(* IEC 61131-3 sources: elnaProjects/ElpcLogic/PomarKc7Changed/build_USO_ecl (part 3) *)

  IM_SingleSignals_dP_maslo_gaz_Less100_status := DWORD_TO_UDINT(Im.SingleSignals.dP_maslo_gaz_Less100.status);

  IM_SingleSignals_dp_kran1_Less100_status := DWORD_TO_UDINT(Im.SingleSignals.dp_kran1_Less100.status);

  IM_SingleSignals_Razreshenie_zagruzki_dvig_status := DWORD_TO_UDINT(Im.SingleSignals.Razreshenie_zagruzki_dvig.status);

  IM_SingleSignals_Vozbud_gotovnost_status := DWORD_TO_UDINT(Im.SingleSignals.Vozbud_gotovnost.status);

  IM_SingleSignals_Vozbud_neispr_tsepey_upr_AVR_pit_status := DWORD_TO_UDINT(Im.SingleSignals.Vozbud_neispr_tsepey_upr_AVR_pit.status);

  IM_SingleSignals_Vozbud_neispravnost_status := DWORD_TO_UDINT(Im.SingleSignals.Vozbud_neispravnost.status);

  IM_SingleSignals_SHAVR1_v_rabote_status := DWORD_TO_UDINT(Im.SingleSignals.SHAVR1_v_rabote.status);

  IM_SingleSignals_SHAVR2_v_rabote_status := DWORD_TO_UDINT(Im.SingleSignals.SHAVR2_v_rabote.status);

  IM_SingleSignals_Avariinoe_otkluch_vikluchatelya_status := DWORD_TO_UDINT(Im.SingleSignals.Avariinoe_otkluch_vikluchatelya.status);

  IM_SingleSignals_Assinhronnii_hod_peregruzka_status := DWORD_TO_UDINT(Im.SingleSignals.Assinhronnii_hod_peregruzka.status);

  IM_SingleSignals_SHU_v_GPA_vkluch_status := DWORD_TO_UDINT(Im.SingleSignals.SHU_v_GPA_vkluch.status);

  IM_SingleSignals_SHP_v_GPA_vkluch_status := DWORD_TO_UDINT(Im.SingleSignals.SHP_v_GPA_vkluch.status);

  IM_SingleSignals_QF1_on_status := DWORD_TO_UDINT(Im.SingleSignals.QF1_on.status);

  IM_SingleSignals_QF2_on_status := DWORD_TO_UDINT(Im.SingleSignals.QF2_on.status);

  IM_SingleSignals_QF23_on_status := DWORD_TO_UDINT(Im.SingleSignals.QF23_on.status);

  IM_SingleSignals_QF4_QF5_on_status := DWORD_TO_UDINT(Im.SingleSignals.QF4_QF5_on.status);

  IM_SingleSignals_QF6_QF7_on_status := DWORD_TO_UDINT(Im.SingleSignals.QF6_QF7_on.status);

  IM_SingleSignals_QF8_QF9_on_status := DWORD_TO_UDINT(Im.SingleSignals.QF8_QF9_on.status);

  IM_SingleSignals_QF10_QF11_on_status := DWORD_TO_UDINT(Im.SingleSignals.QF10_QF11_on.status);

  IM_SingleSignals_QF12_QF13_on_status := DWORD_TO_UDINT(Im.SingleSignals.QF12_QF13_on.status);

  IM_SingleSignals_QF14_QF15_on_status := DWORD_TO_UDINT(Im.SingleSignals.QF14_QF15_on.status);

  IM_SingleSignals_QF22_on_status := DWORD_TO_UDINT(Im.SingleSignals.QF22_on.status);

  IM_SingleSignals_NS_G1_G2_status := DWORD_TO_UDINT(Im.SingleSignals.NS_G1_G2.status);

  IM_SingleSignals_NS_G3_G4_status := DWORD_TO_UDINT(Im.SingleSignals.NS_G3_G4.status);

  IM_SingleSignals_NS_G15_G16_status := DWORD_TO_UDINT(Im.SingleSignals.NS_G15_G16.status);

  IM_SingleSignals_NS_G17_status := DWORD_TO_UDINT(Im.SingleSignals.NS_G17.status);

  IM_SingleSignals_NS_G5_G6_status := DWORD_TO_UDINT(Im.SingleSignals.NS_G5_G6.status);

  IM_SingleSignals_NS_G7_G8_status := DWORD_TO_UDINT(Im.SingleSignals.NS_G7_G8.status);

  IM_SingleSignals_NS_G18_G19_status := DWORD_TO_UDINT(Im.SingleSignals.NS_G18_G19.status);

  IM_SingleSignals_NS_G10_G11_status := DWORD_TO_UDINT(Im.SingleSignals.NS_G10_G11.status);

  IM_SingleSignals_NS_G13_G14_status := DWORD_TO_UDINT(Im.SingleSignals.NS_G13_G14.status);

  IM_SingleSignals_Uroven_masla_akkum_status := DWORD_TO_UDINT(Im.SingleSignals.Uroven_masla_akkum.status);

  IM_SingleSignals_NKU1_GPA_on_status := DWORD_TO_UDINT(Im.SingleSignals.NKU1_GPA_on.status);

  IM_SingleSignals_NKU2_GPA_on_status := DWORD_TO_UDINT(Im.SingleSignals.NKU2_GPA_on.status);

  IM_SingleSignals_AO_KC_ot_SHKS_status := DWORD_TO_UDINT(Im.SingleSignals.AO_KC_ot_SHKS.status);

  IM_SingleSignals_AO_GPA_ot_SHU_status := DWORD_TO_UDINT(Im.SingleSignals.AO_GPA_ot_SHU.status);

  IM_SingleSignals_BEAO_srabotal_status := DWORD_TO_UDINT(Im.SingleSignals.BEAO_srabotal.status);

  IM_SingleSignals_Chastotny_pusk_status := DWORD_TO_UDINT(Im.SingleSignals.Chastotny_pusk.status);

  IM_SingleSignals_Neuspesh_chastotny_pusk_status := DWORD_TO_UDINT(Im.SingleSignals.Neuspesh_chastotny_pusk.status);

  IM_SingleSignals_Rezhim_ruchnogo_regulirovaniya_status := DWORD_TO_UDINT(Im.SingleSignals.Rezhim_ruchnogo_regulirovaniya.status);

  IM_SingleSignals_Osnovnoy_regul_off_status := DWORD_TO_UDINT(Im.SingleSignals.Osnovnoy_regul_off.status);

  IM_SingleSignals_Voltage_sekcii_norm_status := DWORD_TO_UDINT(Im.SingleSignals.Voltage_sekcii_norm.status);

  IM_SingleSignals_Reactorny_pusk_status := DWORD_TO_UDINT(Im.SingleSignals.Reactorny_pusk.status);

  IM_SingleSignals_NO_GPA_ot_SHU_status := DWORD_TO_UDINT(Im.SingleSignals.NO_GPA_ot_SHU.status);

  IM_SingleSignals_AO_GPA_ot_PRU_status := DWORD_TO_UDINT(Im.SingleSignals.AO_GPA_ot_PRU.status);

  IM_SingleSignals_Nalichie_BP1_status := DWORD_TO_UDINT(Im.SingleSignals.Nalichie_BP1.status);

  IM_SingleSignals_Nalichie_BP2_status := DWORD_TO_UDINT(Im.SingleSignals.Nalichie_BP2.status);

  IM_SingleSignals_Nalichie_BP3_status := DWORD_TO_UDINT(Im.SingleSignals.Nalichie_BP3.status);

  IM_SingleSignals_Nalichie_BP4_status := DWORD_TO_UDINT(Im.SingleSignals.Nalichie_BP4.status);

  IM_SingleSignals_Nalichie_BP5_status := DWORD_TO_UDINT(Im.SingleSignals.Nalichie_BP5.status);

  IM_SingleSignals_Nalichie_BP6_status := DWORD_TO_UDINT(Im.SingleSignals.Nalichie_BP6.status);

  IM_SingleSignals_Nalichie_BP7_BP8_status := DWORD_TO_UDINT(Im.SingleSignals.Nalichie_BP7_BP8.status);

  IM_SingleSignals_Nalichie_BP9_BP10_status := DWORD_TO_UDINT(Im.SingleSignals.Nalichie_BP9_BP10.status);

  IM_SingleSignals_Nalichie_cepei_upravlen_mv_status := DWORD_TO_UDINT(Im.SingleSignals.Nalichie_cepei_upravlen_mv.status);

  IM_SingleSignals_Nalichie_220BEAO_status := DWORD_TO_UDINT(Im.SingleSignals.Nalichie_220BEAO.status);

  IM_SingleSignals_Nalichie_per_220_na_vhode_status := DWORD_TO_UDINT(Im.SingleSignals.Nalichie_per_220_na_vhode.status);

  IM_SingleSignals_Nalichie_post_220_na_vhode_status := DWORD_TO_UDINT(Im.SingleSignals.Nalichie_post_220_na_vhode.status);

  IM_SingleSignals_Nalichie_BP11_status := DWORD_TO_UDINT(Im.SingleSignals.Nalichie_BP11.status);

  IM_SingleSignals_Nalichie_BP12_status := DWORD_TO_UDINT(Im.SingleSignals.Nalichie_BP12.status);

  IM_SingleSignals_Dver_SHU_pered_otkrita_status := DWORD_TO_UDINT(Im.SingleSignals.Dver_SHU_pered_otkrita.status);

  IM_SingleSignals_Dver_SHU_zad_otkrita_status := DWORD_TO_UDINT(Im.SingleSignals.Dver_SHU_zad_otkrita.status);

  IM_SingleSignals_EO_GPA_ot_knopki_SHU_status := DWORD_TO_UDINT(Im.SingleSignals.EO_GPA_ot_knopki_SHU.status);

  IM_SingleSignals_EO_EGPA_ot_PRY_status := DWORD_TO_UDINT(Im.SingleSignals.EO_EGPA_ot_PRY.status);

  IM_SingleSignals_Synchroniz_rezhima_K1_status := DWORD_TO_UDINT(Im.SingleSignals.Synchroniz_rezhima_K1.status);

  IM_SingleSignals_Potok_ms_posle_AVOM_status := DWORD_TO_UDINT(Im.SingleSignals.Potok_ms_posle_AVOM.status);

  IM_Kran1_status := DWORD_TO_UDINT(Im.Kran1.status);

  IM_Kran2_status := DWORD_TO_UDINT(Im.Kran2.status);

  IM_Kran3_status := DWORD_TO_UDINT(Im.Kran3.status);

  IM_Kran3b_status := DWORD_TO_UDINT(Im.Kran3b.status);

  IM_Kran4_status := DWORD_TO_UDINT(Im.Kran4.status);

  IM_Kran5_status := DWORD_TO_UDINT(Im.Kran5.status);

  IM_Kran6_status := DWORD_TO_UDINT(Im.Kran6.status);

  IM_nu1_status := DWORD_TO_UDINT(Im.nu1.status);

  IM_nu2_status := DWORD_TO_UDINT(Im.nu2.status);

  IM_pns_status := DWORD_TO_UDINT(Im.pns.status);

  IM_v1_Avom_status := DWORD_TO_UDINT(Im.v1_Avom.status);

  IM_v2_Avom_status := DWORD_TO_UDINT(Im.v2_Avom.status);

  IM_v3_Avom_status := DWORD_TO_UDINT(Im.v3_Avom.status);

  IM_v4_Avom_status := DWORD_TO_UDINT(Im.v4_Avom.status);

  IM_mv_status := DWORD_TO_UDINT(Im.mv.status);

  IM_KaloriferAVOM_status := DWORD_TO_UDINT(Im.KaloriferAVOM.status);

  IM_CMN_status := DWORD_TO_UDINT(Im.CMN.status);

  IM_TEN_kollectora_status := DWORD_TO_UDINT(Im.TEN_kollectora.status);

  IM_TEN_MB_status := DWORD_TO_UDINT(Im.TEN_MB.status);
END_FUNCTION_BLOCK

FUNCTION_BLOCK fb_RashodAlg
  VAR_INPUT
    P_gasIn : struct_AI;
  END_VAR
  VAR_IN_OUT
    StrAi : struct_AI;
  END_VAR
  VAR_INPUT
    T_gasIn : struct_AI;
    dP_konf : struct_AI;
    K : struct_AnalogParametr;
    A : struct_AnalogParametr;
    y0 : struct_AnalogParametr;
  END_VAR
  VAR
    num : LREAL;
    den : LREAL;
    _statusAi : TYPE_StatusAi;
  END_VAR
  VAR CONSTANT
    P0 : LREAL          := 0.1033;
    T0 : LREAL          := 293.0;
  END_VAR

  strAI.opcCommandsDisabled := strAI.inopcCommandsDisabled ;

  IF (P_gasIn.interval < _statusAi.normal) OR
     (T_gasIn.interval < _statusAi.normal) OR
     (dP_konf.interval < _statusAi.normal) THEN
  	StrAi.interval := _statusAi.NOTRELIABLE;
            strAI.status := 	SHL(BOOL_TO_DWORD(strAI.OpcCommandsDisabled ), 21)
  	OR BYTE_TO_DWORD(strAI.interval);
  	RETURN;
  END_IF;

  IF (P_gasIn.value <0.3) THEN
  	StrAi.interval := _statusAi.normal;
  	StrAi.value:= 0.0;
            strAI.status := 	SHL(BOOL_TO_DWORD(strAI.OpcCommandsDisabled ), 21)
  	OR BYTE_TO_DWORD(strAI.interval);
  	RETURN;
  END_IF;

  StrAi.interval:= _statusAi.normal;

  num:= (dP_konf.Value/1000.0)*(T_gasIn.value+273.0)*P0*735.56*K.Value;
  den:= y0.Value*P_gasIn.value*T0 ;

  StrAi.value:= A.Value*SQRT(num/den);

  strAI.status := 	SHL(BOOL_TO_DWORD(strAI.OpcCommandsDisabled ), 21) (* Управление в ВУ заблокировано *)
  		OR BYTE_TO_DWORD(strAI.interval);	              (* интервал *)
END_FUNCTION_BLOCK

FUNCTION_BLOCK fb_Question
  VAR_IN_OUT
    StrQ : struct_Question;
  END_VAR
  VAR
    Asked : UINT;
    _answers : TYPE_Answers;
    _sunpackerCommand : fb_sunpackerCommand;
    source : BYTE;
    parametr : BYTE;
    lastParametr : BYTE;
    cmd : BYTE;
    source_for_Status : BYTE;
    cmd_for_Status : BYTE;
    command_error_for_Status : BYTE;
    resetCmdTimer : TON;
    resetCmdTimerPriznak : BOOL;
    reset_Trig : R_TRIG;
  END_VAR
  VAR CONSTANT
    cmd_answer : UINT          := 1;
  END_VAR

  StrQ.OpcCommandsDisabled := StrQ.inopcCommandsDisabled;

  IF StrQ.ask THEN
  StrQ.inopcCommandsDisabled:=FALSE;
      IF Asked=0 THEN
  	Asked:=StrQ.AnswerVariants;
  	StrQ.answer:=_answers.ANS_NONE;
      END_IF;

      _sunpackerCommand(command := StrQ.inCommand);
  	source := _sunpackerCommand.source;
            parametr := _sunpackerCommand.parametr;
  	cmd := _sunpackerCommand.cmd;

      IF cmd <> 0 AND lastParametr <> parametr AND ((NOT StrQ.OpcCommandsDisabled) AND source > 0)  then
  	CASE BYTE_TO_INT(cmd) OF
  	                               1 :

  				IF Asked<>0 THEN
                                             (* CASE BYTE_TO_INT(parametr) OF
                                              1: answer:=_answers.ANS_YES;
                                              2: answer:=_answers.ANS_NO;
                                              4: answer:=_answers.ANS_CANCEL;
                                              8: answer:=_answers.ANS_RETRY;
  	                                  END_CASE;*)
                                          StrQ.answer:=BYTE_TO_UINT(parametr);
                                          command_error_for_Status := 0;
                                          ELSE
  	                              command_error_for_Status := cmd;
                                          END_IF;
  	END_CASE;
  	source_for_Status := source;
  	cmd_for_Status := cmd;
  	resetCmdTimer(IN := FALSE);
  	resetCmdTimerPriznak := TRUE;
      END_IF;

      lastParametr := parametr;

      resetCmdTimer(IN := resetCmdTimerPriznak, PT := T#5S);
      IF resetCmdTimer.Q THEN
  	resetCmdTimerPriznak := FALSE;
  	source_for_Status := 0;
  	cmd_for_Status := 0;
  	command_error_for_Status := 0;
      END_IF;
  END_IF;

  reset_Trig(CLK := StrQ.reset);
  IF reset_Trig.Q THEN
  	Asked:=0;
  	StrQ.answer:=0;
            StrQ.ask:=FALSE;
            StrQ.reset:=FALSE;
  	StrQ.inopcCommandsDisabled:=TRUE;
  END_IF;

  StrQ.status := SHL(BYTE_TO_DWORD(source_for_Status), 29)
  			OR SHL(BYTE_TO_DWORD(cmd_for_Status), 26)
  			OR SHL(BYTE_TO_DWORD(command_error_for_Status), 23)
  			OR SHL(BOOL_TO_DWORD(StrQ.OpcCommandsDisabled ), 21);
  IF StrQ.answer = 0 THEN
      StrQ.status := StrQ.status  OR SHL(UINT_TO_DWORD(asked), 6);
  ELSE
      StrQ.status := StrQ.status  OR SHL(UINT_TO_DWORD(StrQ.answer), 6);
  END_IF;
END_FUNCTION_BLOCK

FUNCTION_BLOCK fb_ph_AIprotection
  VAR_IN_OUT
    StrAiP : struct_AiProtection;
  END_VAR
  VAR_INPUT
    act : TYPE_PhaseAlgoritmAction;
    PhaseNumber : UINT;
  END_VAR
  VAR_IN_OUT
    StrPh : struct_PhaseAlgoritm;
  END_VAR
  VAR
    CommandFault_Trig : R_TRIG;
    reset_Trig : R_TRIG;
    _statusDualInput : TYPE_statusDualInput;
  END_VAR

  IF StrPh.run AND NOT StrPh.start THEN
  	StrPh.start := TRUE;
  	StrPh.top := FALSE;
  	StrPh.error := FALSE;
            StrPh.run:=FALSE;

  	CASE act OF
  		(*PhaseAlgoritmAction.run*)    _run : runAiProtection(StrAiP); (*cmd_run*)
  		(*PhaseAlgoritmAction.reset*)_reset : resetAiProtection(StrAiP); (*cmd_reset*)
  	END_CASE;
  END_IF;

  IF StrPh.start AND NOT StrPh.top THEN
                      CommandFault_Trig(CLK := StrAiP.hasError);
                      IF CommandFault_Trig.Q THEN
  	          StrPh.error := TRUE;
                      END_IF;

  		CASE act OF
  		(*PhaseAlgoritmAction.run*)    _run:    StrPh.top:=StrAiP.isRunning;

  		(*PhaseAlgoritmAction.reset*) _reset:   StrPh.top := NOT StrAiP.isRunning;
  		END_CASE;

  END_IF;

  IF StrPh.top THEN
  StrPh.error := FALSE;
  END_IF;

  reset_Trig(CLK := StrPh.reset);
  IF reset_Trig.Q THEN
            StrPh.start := FALSE;
  	StrPh.error := FALSE;
  	StrPh.top := FALSE;
            StrPh.run:=FALSE;
            StrPh.reset:=FALSE;
  END_IF;

  StrPh.startStatus := SHL(BOOL_TO_DWORD(StrPh.start), PhaseNumber);
  StrPh.errorStatus := SHL(BOOL_TO_DWORD(StrPh.error), PhaseNumber);
  StrPh.topStatus := SHL(BOOL_TO_DWORD(StrPh.top), PhaseNumber);
END_FUNCTION_BLOCK

FUNCTION_BLOCK fb_OilPump_Init
  VAR_INPUT
    data_Ini : BOOL;
    ISVALIDREF_statOn : BOOL;
    ISVALIDREF_statOff : BOOL;
    ISVALIDREF_cmdOn : BOOL;
    ISVALIDREF_cmdOff : BOOL;
    ISVALIDREF_inBreakCmdOn : BOOL;
    ISVALIDREF_inBreakCmdOff : BOOL;
  END_VAR
  VAR_IN_OUT
    str_Op : struct_OilPump;
  END_VAR
  VAR_OUTPUT
    Init : BOOL          := FALSE;
  END_VAR

  (*****            Функциональный блок переинициализации структуры  НУ          *****)

   Init := FALSE;

      IF data_Ini THEN                            (* Параметрам требуется переинициализация. *)
          str_Op.ISVALIDREF_statOn                := ISVALIDREF_statOn;
          str_Op.ISVALIDREF_statOff               := ISVALIDREF_statOff;
          str_Op.ISVALIDREF_cmdOn                 := ISVALIDREF_cmdOn;
          str_Op.ISVALIDREF_cmdOff                := ISVALIDREF_cmdOff;
          str_Op.ISVALIDREF_inBreakCmdOn          := ISVALIDREF_inBreakCmdOn;
          str_Op.ISVALIDREF_inBreakCmdOff         := ISVALIDREF_inBreakCmdOff;
          data_Ini:=FALSE;
          Init := TRUE;
      END_IF;

          ISVALIDREF_statOn:= FALSE;
          ISVALIDREF_statOff:= FALSE;
          ISVALIDREF_cmdOn:= FALSE;
          ISVALIDREF_cmdOff:= FALSE;
          ISVALIDREF_inBreakCmdOn:= FALSE;
          ISVALIDREF_inBreakCmdOff:= FALSE;
END_FUNCTION_BLOCK

FUNCTION_BLOCK fb_DO_Init
  VAR_INPUT
    data_Ini : BOOL;
    imit : BOOL          := FALSE;
  END_VAR
  VAR_IN_OUT
    strDO : struct_DO;
  END_VAR
  VAR_OUTPUT
    Init : BOOL          := FALSE;
  END_VAR

  (*****            Функциональный блок переинициализации структуры-дескриптора канала дискретного ввода.            *****)
   Init := FALSE;

      IF data_Ini THEN                            (* Параметрам требуется переинициализация. *)
          strDO.imit       := imit;
          data_Ini:=FALSE;
          Init := TRUE;
      END_IF;
    IF Init THEN
  imit:=FALSE;
     END_IF;
END_FUNCTION_BLOCK

FUNCTION_BLOCK fb_DOSourceMlp
  VAR_IN_OUT
    arDout : TWordData;
  END_VAR
  VAR_INPUT
    err_mod : TItemDIN;
  END_VAR
  VAR_IN_OUT
    strDO : struct_DO;
  END_VAR
  VAR
    bitNumber : INT;
  END_VAR

  strDO.blConnect := ((UINT_TO_WORD(err_mod.wValue) = 20) and (UINT_TO_WORD(err_mod.wFlags) = 192));

  strDO.value:=0;

  FOR bitNumber:=0 TO 15 BY 1 DO
  	strDO.value:=strDO.value OR (SHL(BOOL_TO_WORD(strDO.bits[bitNumber]),bitNumber));
  END_FOR;

  IF NOT strDO.imit THEN
  	 arDout.wValue:= WORD_TO_UINT(strDO.value);
  END_IF;
END_FUNCTION_BLOCK

FUNCTION_BLOCK fb_AnalogParametr
  VAR_IN_OUT
    StrAP : struct_AnalogParametr;
  END_VAR
  VAR
    _sunpackerCommand : fb_sunpackerCommand;
    source : BYTE;
    cmd : BYTE;
    source_for_Status : BYTE;
    cmd_for_Status : BYTE;
    command_error_for_Status : BYTE;
    resetCmdTimer : TON;
    resetCmdTimerPriznak : BOOL;
    secondTact : BOOL;
    inp : LREAL;
    rABS : LREAL;
  END_VAR

  IF NOT secondTact THEN
  	StrAP.Value := StrAP.currentValue;
  	secondTact := true;
  END_IF;

  StrAP.OpcCommandsDisabled := StrAP.inOpcCommandsDisabled;

   (* ---- Если управление с ВУ заблокировано, то передаем команду из алгоритма ---- *)
  IF StrAP.inOpcCommandsDisabled THEN
  	StrAP.inCommand := StrAP.inCommand_Alg;
  ELSE (* иначе передаем команду с АРМа*)
  	StrAP.inCommand := StrAP.inCommand_ARM;
  END_IF;

  _sunpackerCommand(command := StrAP.inCommand);
  	source := _sunpackerCommand.source;
  	cmd := _sunpackerCommand.cmd;

  IF cmd <> 0 AND StrAP.newValue <> StrAP.Value and (((NOT StrAP.opcCommandsDisabled) AND source > 0) OR source = 0) then
  	CASE BYTE_TO_INT(cmd) OF
  	(*cmd_ChangeValue*) 1 :
  				StrAP.isValidValue := TRUE;
  				IF StrAP.minVal_ISVALIDREF AND StrAP.isValidValue THEN
  					IF StrAP.newValue < StrAP.minVal THEN
  						StrAP.isValidValue := FALSE;
  					END_IF;
  				END_IF;
  				IF StrAP.maxVal_ISVALIDREF AND StrAP.isValidValue THEN
  					IF StrAP.newValue > StrAP.maxVal THEN
  						StrAP.isValidValue := FALSE;
  					END_IF;
  				END_IF;
  				IF StrAP.maxStep_ISVALIDREF AND StrAP.isValidValue  THEN
  					inp := StrAP.Value - StrAP.newValue;
  					IF inp < 0.0 THEN
  						rABS := -inp;
  					ELSE
  						rABS := inp;
  					END_IF;
  					IF rABS > StrAP.maxStep THEN
  						StrAP.isValidValue := FALSE;
  					END_IF;
  				END_IF;
  				IF StrAP.isValidValue THEN
  					StrAP.Value := StrAP.newValue;
  					command_error_for_Status := 0;
  				ELSE
  					command_error_for_Status := cmd;
  				END_IF;
  	END_CASE;
  	source_for_Status := source;
  	cmd_for_Status := cmd;
  	resetCmdTimer(IN := FALSE);
  	resetCmdTimerPriznak := TRUE;
  END_IF;

  resetCmdTimer(IN := resetCmdTimerPriznak, PT := T#5S);
  IF resetCmdTimer.Q THEN
  	resetCmdTimerPriznak := FALSE;
  	source_for_Status := 0;
  	cmd_for_Status := 0;
  	command_error_for_Status := 0;
  END_IF;

  StrAP.status := SHL(BYTE_TO_DWORD(source_for_Status), 29)
  			OR SHL(BYTE_TO_DWORD(cmd_for_Status), 26)
  			OR SHL(BYTE_TO_DWORD(command_error_for_Status), 23)
  			OR SHL(BOOL_TO_DWORD(StrAP.OpcCommandsDisabled ), 21);
END_FUNCTION_BLOCK

FUNCTION_BLOCK fb_AI_Init
  VAR_INPUT
    data_Ini : BOOL;
    dLL : LREAL;
    dHL : LREAL;
    dLA : LREAL;
    dHA : LREAL;
    dLW : LREAL;
    dHW : LREAL;
    ISVALIDREF_LA : BOOL          := False;
    ISVALIDREF_HA : BOOL          := False;
    ISVALIDREF_LW : BOOL          := False;
    ISVALIDREF_HW : BOOL          := False;
    delayLA : TIME          := T#0S;
    delayLW : TIME          := T#0S;
    delayHW : TIME          := T#0S;
    delayHA : TIME          := T#0S;
    inpLL : LREAL          := 4000.0;
    inpHL : LREAL          := 20000.0;
    CurrentShotCircuit : LREAL          := 21000.0;
    CurrentBreakCircuit : LREAL          := 3700.0;
    dMaxChangeSpeed : LREAL;
    dMaxChangeSpeedDown : LREAL;
    histeresis : LREAL;
    aperturFilter : LREAL;
    exponentialFilter : LREAL;
    rassoglasovanie : LREAL;
    inOpcCommandsDisabled : BOOL;
  END_VAR
  VAR_IN_OUT
    strAI : struct_AI;
  END_VAR
  VAR_OUTPUT
    Init : BOOL          := FALSE;
  END_VAR

  (*****            Функциональный блок переинициализации структуры-дескриптора канала аналогового ввода.            *****)
       Init := false;

      IF data_Ini THEN                            (* Параметрам требуется переинициализация. *)
          strAI.dLL                := dLL;
          strAI.dHL                := dHL;
          strAI.dLA                := dLA;
          strAI.dHA                := dHA;
          strAI.dLW                := dLW;
          strAI.dHW                := dHW;
          strAI.ISVALIDREF_LA      := ISVALIDREF_LA;
          strAI.ISVALIDREF_HA      := ISVALIDREF_HA;
          strAI.ISVALIDREF_LW      := ISVALIDREF_LW;
          strAI.ISVALIDREF_HW      := ISVALIDREF_HW;
          strAI.delayLA            := delayLA;
          strAI.delayLW            := delayLW;
          strAI.delayHW            := delayHW;
          strAI.delayHA            := delayHA;
          strAI.inpLL              := inpLL;
          strAI.inpHL              := inpHL;
          strAI.CurrentShotCircuit := CurrentShotCircuit;
          strAI.CurrentBreakCircuit:= CurrentBreakCircuit;
          strAI.dMaxChangeSpeed     := dMaxChangeSpeed;
          strAI.dMaxChangeSpeedDown := dMaxChangeSpeedDown;
          strAI.histeresis         := histeresis;
          strAI.aperturFilter      := aperturFilter;
          strAI.exponentialFilter  := exponentialFilter;
          strAI.rassoglasovanie    := rassoglasovanie;
          strAI.rassoglasovanie    := rassoglasovanie;

          data_Ini:=false;
          Init := TRUE;
       END_IF;
    IF Init THEN
          dLL:= 0.0;
          dHL:= 0.0;
          dLA:= 0.0;
          dHA:= 0.0;
          dLW:= 0.0;
          dHW:= 0.0;
          inpLL:= 4000.0;
          inpHL:= 20000.0;
          CurrentShotCircuit:= 21000.0;
          CurrentBreakCircuit:= 3700.0;
          ISVALIDREF_LA:= false;
          ISVALIDREF_HA:= false;
          ISVALIDREF_LW:= false;
          ISVALIDREF_HW:= false;
          delayLA:= T#0S;
          delayLW:= T#0S;
          delayHW:= T#0S;
          delayHA:= T#0S;
          dMaxChangeSpeed:= 0.0;
          dMaxChangeSpeedDown:= 0.0;
          histeresis:= 0.0;
          aperturFilter:= 0.0;
          exponentialFilter:= 0.0;
          rassoglasovanie:= 0.0;
        END_IF;
END_FUNCTION_BLOCK

FUNCTION_BLOCK fb_AiSourceMlp_timer
  VAR_INPUT
    arAIN : TItemAIN;
    err_mod : TItemDIN;
  END_VAR
  VAR_IN_OUT
    strAI : struct_AI;
  END_VAR
  VAR
    _statusAi : TYPE_StatusAi;
    _commandAnalog : TYPE_CommandAnalog;
    _sunpackerCommand : fb_sunpackerCommand;
    _AnalogLimitFlags : TYPE_AnalogLimitFlags;
    notReliable : BOOL;
    _lastValue : LREAL;
    resetCmdTimer : TON;
    _LastValueTimer : TON;
    resetCmdTimerPriznak : BOOL;
    k : LREAL;
    b : LREAL;
    ap : LREAL;
    raznitsa : LREAL;
    rABS : LREAL;
    h : LREAL;
    mismatch : LREAL;
    parametr : BYTE;
    source : BYTE;
    cmd : BYTE;
    lastCmd : BYTE;
    source_for_Status : BYTE;
    cmd_for_Status : BYTE;
    command_error_for_Status : BYTE;
    secondTakt : BOOL;
    off_trig : R_TRIG;
    on_trig : R_TRIG;
    remont_trig : R_TRIG;
    LL_trig : R_TRIG;
    HL_trig : R_TRIG;
    Normal_trig : R_TRIG;
    Nedostover_trig : R_TRIG;
    timerLA : TON;
    timerHA : TON;
    timerLW : TON;
    timerHW : TON;
  END_VAR
  VAR RETAIN
    retainLL : LREAL;
    retainHL : LREAL;
    retainLA : LREAL;
    retainHA : LREAL;
    retainLW : LREAL;
    retainHW : LREAL;
  END_VAR

  strAI.opcCommandsDisabled := strAI.inopcCommandsDisabled ;

  (* ---- При первом пуске принимаем значение уставок ---- *)
  IF NOT secondTakt THEN
            IF (strAI.dLL <> retainLL) AND (retainLL <> 0.0) THEN  strAI.LL := retainLL;
            ELSE strAI.LL := strAI.dLL; END_IF;
  	IF (strAI.dHL <> retainHL) AND (retainHL <> 0.0) THEN  strAI.HL := retainHL;
            ELSE strAI.HL := strAI.dHL; END_IF;

            IF strAI.ISVALIDREF_HA AND (strAI.dHA <> retainHA) AND (retainHA <> 0.0) THEN  strAI.HA := retainHA;
            ELSE strAI.HA := strAI.dHA; END_IF;

            IF strAI.ISVALIDREF_LA AND (strAI.dLA <> retainLA) AND (retainLA <> 0.0) THEN  strAI.LA := retainLA;
            ELSE strAI.LA := strAI.dLA; END_IF;

            IF strAI.ISVALIDREF_HW AND (strAI.dHW <> retainHW) AND (retainHW <> 0.0) THEN  strAI.HW := retainHW;
            ELSE strAI.HW := strAI.dHW; END_IF;

            IF strAI.ISVALIDREF_LW AND (strAI.dLW <> retainLW) AND (retainLW <> 0.0) THEN  strAI.LW := retainLW;
            ELSE strAI.LW := strAI.dLW; END_IF;

  	secondTakt  := TRUE;
  END_IF;

  (* ---- пересчет тока в физ величину ---- *)
  k := (strAI.HL - strAI.LL)/(strAI.inpHl - strAI.inpLL);
  b := strAI.LL - k * strAI.inpLL;
  strAI.value := k * arAIN.dblValue + b;

  (* ---- определение обрыва и кз ----- *)

  strAI.blConnect := true;(*(UINT_TO_WORD(arAIN.wFlags) = 1472) and (UINT_TO_WORD(err_mod.wValue) = 20) and (UINT_TO_WORD(err_mod.wFlags) = 192); *)
  IF NOT strAI.blConnect THEN
      strAI.interval := _statusAi.NOTDEFINED;
  ELSIF ((arAIN.dblValue < strAI.currentBreakCircuit) AND (strAI.currentBreakCircuit > 0.0)) OR ((strAI.interval = _statusAi.LL) AND (arAIN.dblValue < (strAI.currentBreakCircuit + 100.0))) THEN
      strAI.interval := _statusAi.LL;
  ELSIF ((arAIN.dblValue > strAI.currentShotCircuit) AND (strAI.currentShotCircuit > 0.0)) OR ((strAI.interval = _statusAi.HL) AND (arAIN.dblValue > (strAI.currentShotCircuit - 100.0))) THEN
      strAI.interval := _statusAi.HL;
  ELSE
      strAI.interval := _statusAi.normal;
  END_IF;

  IF NOT strAI.imit THEN
  	(* Расчет апертурного фильтра*)
  	ap := strAI.aperturFilter * 0.01 * (strAI.HL - strAI.LL);
  	IF strAI.aperturFilter <> 0.0 THEN raznitsa := strAI.value- _lastValue;
  		IF 	raznitsa < 0.0 	THEN 	rABS := -raznitsa; 		ELSE 	rABS := raznitsa; 		END_IF;
  		IF 	rABS > ap 	THEN 	strAI.value := strAI.value;	ELSE 	strAI.value := _lastValue; 	END_IF;
  	END_IF;

  	(* Расчет экпоненциального фильтра*)
  	IF strAI.exponentialFilter <> 0.0 THEN strAI.value := (strAI.exponentialFilter * strAI.value) + ((1.0 - strAI.exponentialFilter) * _lastValue); END_IF;
  ELSE
  	strAI.interval := _statusAi.normal;
  END_IF;

  IF notReliable THEN strAI.interval := _statusAi.NOTRELIABLE; END_IF;

  IF NOT notReliable THEN
  	IF strAI.interval >= _statusAi.normal THEN
  		strAI.interval := _statusAi.NOTDEFINED;
  		h := strAI.histeresis* 0.01 * (strAI.HL-strAI.LL);
  		(*определение выхода за аппаратные границы вынесено в GetData.здесь только для нужд имитации*)
  		IF strAI.imit THEN
  			mismatch := strAI.rassoglasovanie * 0.01 * (strAI.HL - strAI.LL);
  			IF ( strAI.value < strAI.LL - mismatch)   THEN strAI.interval := _statusAi.LL;
  			ELSIF  (strAI.value > strAI.Hl + mismatch) THEN strAI.interval := _statusAi.HL; END_IF;
  		ELSE
  			strAI.interval := _statusAi.normal;
  			IF strAI.ISVALIDREF_LA AND NOT strAI.Disabled_LA AND (strAI.interval = _statusAi.normal) THEN
                                timerLA(IN:=(strAI.value  < strAI.LA) OR ((strAI.interval = _statusAi.LA)  AND ((strAI.value - h) < strAI.LA)), PT:=strAI.delayLA);
  				IF timerLA.Q  THEN
  					strAI.interval := _statusAi.LA;
  				END_IF;
  			END_IF;
  			IF strAI.ISVALIDREF_HA  AND NOT strAI.Disabled_HA AND (strAI.interval = _statusAi.normal)  THEN
                                timerHA(IN:=(strAI.value > strAI.HA) OR ((strAI.interval = _statusAi.HA)  AND ((strAI.value + h) > strAI.HA)), PT:=strAI.delayHA);
  				IF timerHA.Q  THEN
  					strAI.interval := _statusAi.HA;
  				END_IF;
  			END_IF;
  			IF strAI.ISVALIDREF_LW AND NOT strAI.Disabled_LW AND (strAI.interval = _statusAi.normal)  THEN
                                timerLW(IN:=(strAI.value < strAI.LW) OR ((strAI.interval = _statusAi.LW)  AND ((strAI.value - h) < strAI.LW)), PT:=strAI.delayLW);
  				IF timerLW.Q THEN
  					strAI.interval := _statusAi.LW;
  				END_IF;
  			END_IF;
  			IF strAI.ISVALIDREF_HW AND NOT strAI.Disabled_HW  AND (strAI.interval = _statusAi.normal) THEN
                                timerHW(IN:=(strAI.value > strAI.HW)  OR ((strAI.interval = _statusAi.HW)  AND ((strAI.value + h) > strAI.HW)), PT:=strAI.delayHW);
  				IF  timerHW.Q  THEN
  					strAI.interval := _statusAi.HW;
  				END_IF;
  			END_IF;
  		END_IF;
  	END_IF;
  ELSE
  	strAI.interval := _statusAi.NOTRELIABLE;
  END_IF;

  IF strAI.remont THEN strAI.interval := _statusAi.NOTDEFINED; END_IF;

  _sunpackerCommand(command := strAI.inCommand);
  	source := _sunpackerCommand.source;
  	parametr := _sunpackerCommand.parametr;
  	cmd := _sunpackerCommand.cmd;

  IF cmd <> 0 AND lastCmd <> cmd and (((NOT strAI.opcCommandsDisabled) AND source > 0) OR source = 0) then
  	CASE BYTE_TO_INT(cmd) OF
  	(*cmd_SetUstavki*) 1 :
  				IF ((parametr AND _AnalogLimitFlags.LL) <> 0)		             	THEN 	strAI.LL := strAI.dLL; retainLL:= strAI.LL; END_IF;
  				IF ((parametr AND _AnalogLimitFlags.HL) <> 0)		 	          THEN	strAI.HL := strAI.dHL; retainHL:= strAI.HL; END_IF;
  				IF ((parametr AND _AnalogLimitFlags.LA) <> 0) AND strAI.ISVALIDREF_LA 	THEN	strAI.LA := strAI.dLA; retainLA:= strAI.LA; END_IF;
  				IF ((parametr AND _AnalogLimitFlags.HA) <> 0) AND strAI.ISVALIDREF_HA 	THEN	strAI.HA := strAI.dHA; retainHA:= strAI.HA; END_IF;
  				IF ((parametr AND _AnalogLimitFlags.LW) <> 0) AND strAI.ISVALIDREF_LW 	THEN	strAI.LW := strAI.dLW; retainLW:= strAI.LW; END_IF;
  				IF ((parametr AND _AnalogLimitFlags.HW) <> 0) AND strAI.ISVALIDREF_HW 	THEN	strAI.HW := strAI.dHW; retainHW:= strAI.HW; END_IF;
  	(*cmd_SetRemont*) 2 :
  				strAI.remont := TRUE;
  	(*cmd_ResetRemont*) 3 :
  				strAI.remont := FALSE;
  	(*cmd_kvitNotReliable*) 4 :
  				notReliable := FALSE;
  	END_CASE;
  	source_for_Status := source;
  	cmd_for_Status := cmd;
  	command_error_for_Status := 0;
  	resetCmdTimer(IN := FALSE);
  	resetCmdTimerPriznak := TRUE;
  END_IF;
  lastCmd := cmd;

  resetCmdTimer(IN := resetCmdTimerPriznak, PT := T#5S);
  IF resetCmdTimer.Q THEN
  	resetCmdTimerPriznak := FALSE;
  	source_for_Status := 0;
  	cmd_for_Status := 0;
  	command_error_for_Status := 0;
  END_IF;

  strAI.NS_Min := (strAI.value < strAI.minValue) AND strAI.minValue_ISVALIDREF;
  strAI.NS_Max := (strAI.value > strAI.maxValue) AND strAI.maxValue_ISVALIDREF;

  strAI.NS := (strAI.interval <= _statusAi.normal) AND NOT strAI.remont;

  Normal_trig(CLK := strAI.interval >= _statusAi.normal);

  IF NOT Normal_trig.Q THEN
  	_LastValueTimer(PT := T#1S);
  	IF (strAI.value<>_lastValue) OR _LastValueTimer.Q THEN
  		IF (_LastValueTimer.ET>T#0MS) THEN
  			strAI.ChangeSpeed:=(strAI.value-_lastValue)/(TIME_TO_LREAL(_LastValueTimer.ET)/1000.0);
  		END_IF;
  		_LastValueTimer(IN:=FALSE);

  		_LastValueTimer(IN:=TRUE);
  	END_IF;
  END_IF;
  _lastValue := strAI.value;

  IF ((strAI.maxChangeSpeed<>0.0) OR  (strAI.maxChangeSpeedDown<>0.0)) AND ( strAI.interval>=_statusAi.normal) THEN
  		IF (strAI.ChangeSpeed>0.0) THEN
  		    IF (strAI.ChangeSpeed > strAI.maxChangeSpeed) AND (strAI.maxChangeSpeed>0.0000001) THEN
  			 notReliable:=TRUE;
  		    END_IF;
  		ELSE
  		    IF (ABS(strAI.ChangeSpeed)>strAI.maxChangeSpeedDown) AND (strAI.maxChangeSpeedDown>0.0000001)  THEN
                                 notReliable:=TRUE;
  		    END_IF;
  		END_IF;

  END_IF;

  strAI.status := SHL(BYTE_TO_DWORD(source_for_Status), 29) 		              (* Источник команды *)
  			OR SHL(BYTE_TO_DWORD(cmd_for_Status), 26) 	    (* Команда *)
  			OR SHL(BYTE_TO_DWORD(command_error_for_Status), 23)   (* Ошибка команды *)
  			OR SHL(BOOL_TO_DWORD(strAI.OpcCommandsDisabled ), 21) (* Управление в ВУ заблокировано *)
  			OR SHL(BOOL_TO_DWORD(strAI.Disabled_HA), 9)		    (* ВА исключена из формирования интервала *)
  			OR SHL(BOOL_TO_DWORD(strAI.Disabled_LA), 8)		    (* НА исключена из формирования интервала *)
  			OR SHL(BOOL_TO_DWORD(strAI.Disabled_HW), 7)		    (* ВП исключена из формирования интервала *)
  			OR SHL(BOOL_TO_DWORD(strAI.Disabled_LW), 6)	              (* НП исключена из формирования интервала *)
  			OR SHL(BOOL_TO_DWORD(strAI.NS), 5)			    (* неиспарвность сигнала *)
  			OR SHL(BOOL_TO_DWORD(strAI.remont), 4)	              (* Выведен в ремонт *)
  			OR BYTE_TO_DWORD(strAI.interval);	              (* интервал *)
END_FUNCTION_BLOCK

FUNCTION_BLOCK fb_AiSourceMlp
  VAR_INPUT
    arAIN : TItemAIN;
    err_mod : TItemDIN;
  END_VAR
  VAR_IN_OUT
    strAI : struct_AI;
  END_VAR
  VAR
    _statusAi : TYPE_StatusAi;
    _commandAnalog : TYPE_CommandAnalog;
    _sunpackerCommand : fb_sunpackerCommand;
    _AnalogLimitFlags : TYPE_AnalogLimitFlags;
    notReliable : BOOL;
    _lastValue : LREAL;
    resetCmdTimer : TON;
    _LastValueTimer : TON;
    resetCmdTimerPriznak : BOOL;
    k : LREAL;
    b : LREAL;
    ap : LREAL;
    raznitsa : LREAL;
    rABS : LREAL;
    h : LREAL;
    mismatch : LREAL;
    parametr : BYTE;
    source : BYTE;
    cmd : BYTE;
    lastCmd : BYTE;
    source_for_Status : BYTE;
    cmd_for_Status : BYTE;
    command_error_for_Status : BYTE;
    onInit : BOOL;
    off_trig : R_TRIG;
    on_trig : R_TRIG;
    remont_trig : R_TRIG;
    LL_trig : R_TRIG;
    HL_trig : R_TRIG;
    Normal_trig : R_TRIG;
    Nedostover_trig : R_TRIG;
  END_VAR

  strAI.opcCommandsDisabled := strAI.inopcCommandsDisabled ;

  (* ---- При первом пуске принимаем значение уставок ---- *)
  IF NOT onInit THEN

            strAI.LL := strAI.dLL;
            strAI.HL := strAI.dHL;

            strAI.MaxChangeSpeed     := strAI.dMaxChangeSpeed;
            strAI.MaxChangeSpeedDown := strAI.dMaxChangeSpeedDown;

            IF strAI.ISVALIDREF_HA THEN strAI.HA := strAI.dHA; END_IF;

            IF strAI.ISVALIDREF_LA THEN strAI.LA := strAI.dLA; END_IF;

            IF strAI.ISVALIDREF_HW THEN strAI.HW := strAI.dHW; END_IF;

            IF strAI.ISVALIDREF_LW THEN strAI.LW := strAI.dLW; END_IF;

  	onInit  := TRUE;
  END_IF;

  (* ---- пересчет тока в физ величину ---- *)
  k := (strAI.HL - strAI.LL)/(strAI.inpHl - strAI.inpLL);
  b := strAI.LL - k * strAI.inpLL;
  strAI.value := k * arAIN.dblValue + b;

  (* ---- определение обрыва и кз ----- *)

  strAI.blConnect :=(*(UINT_TO_WORD(arAIN.wFlags) = 1472) and*) (UINT_TO_WORD(err_mod.wValue) = 20) and (UINT_TO_WORD(err_mod.wFlags) = 192);
  IF NOT strAI.blConnect THEN
      strAI.interval := _statusAi.NOTDEFINED;
  ELSIF ((arAIN.dblValue < strAI.currentBreakCircuit) AND (strAI.currentBreakCircuit > 0.0)) OR ((strAI.interval = _statusAi.LL) AND (arAIN.dblValue < (strAI.currentBreakCircuit + 100.0))) THEN
      strAI.interval := _statusAi.LL;
  ELSIF ((arAIN.dblValue > strAI.currentShotCircuit) AND (strAI.currentShotCircuit > 0.0)) OR ((strAI.interval = _statusAi.HL) AND (arAIN.dblValue > (strAI.currentShotCircuit - 100.0))) THEN
      strAI.interval := _statusAi.HL;
  ELSE
      strAI.interval := _statusAi.normal;
  END_IF;

  IF NOT strAI.imit THEN
  	(* Расчет апертурного фильтра*)
  	ap := strAI.aperturFilter * 0.01 * (strAI.HL - strAI.LL);
  	IF strAI.aperturFilter <> 0.0 THEN raznitsa := strAI.value- _lastValue;
  		IF 	raznitsa < 0.0 	THEN 	rABS := -raznitsa; 		ELSE 	rABS := raznitsa; 		END_IF;
  		IF 	rABS > ap 	THEN 	strAI.value := strAI.value;	ELSE 	strAI.value := _lastValue; 	END_IF;
  	END_IF;

  	(* Расчет экпоненциального фильтра*)
  	IF strAI.exponentialFilter <> 0.0 THEN strAI.value := (strAI.exponentialFilter * strAI.value) + ((1.0 - strAI.exponentialFilter) * _lastValue); END_IF;
  ELSE
  	strAI.interval := _statusAi.normal;
  END_IF;

  IF notReliable THEN strAI.interval := _statusAi.NOTRELIABLE; END_IF;

  IF NOT notReliable THEN
  	IF strAI.interval >= _statusAi.normal THEN
  		strAI.interval := _statusAi.NOTDEFINED;
  		h := strAI.histeresis* 0.01 * (strAI.HL-strAI.LL);
  		(*определение выхода за аппаратные границы вынесено в GetData.здесь только для нужд имитации*)
  		IF strAI.imit THEN
  			mismatch := strAI.rassoglasovanie * 0.01 * (strAI.HL - strAI.LL);
  			IF ( strAI.value < strAI.LL - mismatch)   THEN strAI.interval := _statusAi.LL;
  			ELSIF  (strAI.value > strAI.Hl + mismatch) THEN strAI.interval := _statusAi.HL; END_IF;
  		ELSE
  			strAI.interval := _statusAi.normal;
  			IF strAI.ISVALIDREF_LA AND NOT strAI.Disabled_LA AND (strAI.interval = _statusAi.normal) THEN
  				IF (strAI.value  < strAI.LA) OR ((strAI.interval = _statusAi.LA)  AND ((strAI.value - h) < strAI.LA))  THEN
  					strAI.interval := _statusAi.LA;
  				END_IF;
  			END_IF;
  			IF strAI.ISVALIDREF_HA  AND NOT strAI.Disabled_HA AND (strAI.interval = _statusAi.normal)  THEN
  				IF (strAI.value > strAI.HA) OR ((strAI.interval = _statusAi.HA)  AND ((strAI.value + h) > strAI.HA))  THEN
  					strAI.interval := _statusAi.HA;
  				END_IF;
  			END_IF;
  			IF strAI.ISVALIDREF_LW AND NOT strAI.Disabled_LW AND (strAI.interval = _statusAi.normal)  THEN
  				IF (strAI.value < strAI.LW) OR ((strAI.interval = _statusAi.LW)  AND ((strAI.value - h) < strAI.LW)) THEN
  					strAI.interval := _statusAi.LW;
  				END_IF;
  			END_IF;
  			IF strAI.ISVALIDREF_HW AND NOT strAI.Disabled_HW  AND (strAI.interval = _statusAi.normal) THEN
  				IF (strAI.value > strAI.HW)  OR ((strAI.interval = _statusAi.HW)  AND ((strAI.value + h) > strAI.HW))   THEN
  					strAI.interval := _statusAi.HW;
  				END_IF;
  			END_IF;
  		END_IF;
  	END_IF;
  ELSE
  	strAI.interval := _statusAi.NOTRELIABLE;
  END_IF;

  IF strAI.remont THEN strAI.interval := _statusAi.NOTDEFINED; END_IF;

  (* ---- Если управление с ВУ заблокировано, то  передаем команду из алгоритма ---- *)
  IF strAI.inOpcCommandsDisabled THEN
  	strAI.inCommand := strAI.inCommand_Alg;
  ELSE (* иначе передаем команду с АРМа*)
  	strAI.inCommand := strAI.inCommand_ARM;
  END_IF;

  _sunpackerCommand(command := strAI.inCommand);
  	source := _sunpackerCommand.source;
  	parametr := _sunpackerCommand.parametr;
  	cmd := _sunpackerCommand.cmd;

  IF cmd <> 0 AND lastCmd <> cmd and (((NOT strAI.opcCommandsDisabled) AND source > 0) OR source = 0) then
  	CASE BYTE_TO_INT(cmd) OF
  	(*cmd_SetUstavki*) 1 :
  				IF ((parametr AND _AnalogLimitFlags.LL) <> 0)		             	THEN 	strAI.LL := strAI.dLL; END_IF;
  				IF ((parametr AND _AnalogLimitFlags.HL) <> 0)		 	          THEN	strAI.HL := strAI.dHL; END_IF;
  				IF ((parametr AND _AnalogLimitFlags.LA) <> 0) AND strAI.ISVALIDREF_LA 	THEN	strAI.LA := strAI.dLA; END_IF;
  				IF ((parametr AND _AnalogLimitFlags.HA) <> 0) AND strAI.ISVALIDREF_HA 	THEN	strAI.HA := strAI.dHA; END_IF;
  				IF ((parametr AND _AnalogLimitFlags.LW) <> 0) AND strAI.ISVALIDREF_LW 	THEN	strAI.LW := strAI.dLW; END_IF;
  				IF ((parametr AND _AnalogLimitFlags.HW) <> 0) AND strAI.ISVALIDREF_HW 	THEN	strAI.HW := strAI.dHW; END_IF;
                                          IF ((parametr AND _AnalogLimitFlags.SipUP) <> 0)                       	THEN	strAI.MaxChangeSpeed     := strAI.dMaxChangeSpeed;     END_IF;
  				IF ((parametr AND _AnalogLimitFlags.SipDown) <> 0)                      	THEN	strAI.MaxChangeSpeedDown := strAI.dMaxChangeSpeedDown; END_IF;

  	(*cmd_SetRemont*) 6 :
  				strAI.remont := TRUE;
  	(*cmd_ResetRemont*) 7 :
  				strAI.remont := FALSE;
  	(*cmd_kvitNotReliable*) 4 :
  				notReliable := FALSE;
  	END_CASE;
  	source_for_Status := source;
  	cmd_for_Status := cmd;
  	command_error_for_Status := 0;
  	resetCmdTimer(IN := FALSE);
  	resetCmdTimerPriznak := TRUE;
  END_IF;
  lastCmd := cmd;

  resetCmdTimer(IN := resetCmdTimerPriznak, PT := T#5S);
  IF resetCmdTimer.Q THEN
  	resetCmdTimerPriznak := FALSE;
  	source_for_Status := 0;
  	cmd_for_Status := 0;
  	command_error_for_Status := 0;
  END_IF;

  strAI.NS_Min := (strAI.value < strAI.minValue) AND strAI.minValue_ISVALIDREF;
  strAI.NS_Max := (strAI.value > strAI.maxValue) AND strAI.maxValue_ISVALIDREF;

  strAI.NS := (strAI.interval <= _statusAi.normal) AND NOT strAI.remont;

  Normal_trig(CLK := strAI.interval >= _statusAi.normal);

  IF NOT Normal_trig.Q THEN
  	_LastValueTimer(PT := T#1S);
  	IF (strAI.value<>_lastValue) OR _LastValueTimer.Q THEN
  		IF (_LastValueTimer.ET>T#0MS) THEN
  			strAI.ChangeSpeed:=(strAI.value-_lastValue)/(TIME_TO_LREAL(_LastValueTimer.ET));
  		END_IF;
  		_LastValueTimer(IN:=FALSE);

  		_LastValueTimer(IN:=TRUE);
  	END_IF;
  END_IF;
  _lastValue := strAI.value;

  IF ((strAI.maxChangeSpeed<>0.0) OR  (strAI.maxChangeSpeedDown<>0.0)) AND ( strAI.interval>=_statusAi.normal) THEN
  		IF (strAI.ChangeSpeed>0.0) THEN
  		    IF (strAI.ChangeSpeed > strAI.maxChangeSpeed) AND (strAI.maxChangeSpeed>0.0000001) THEN
  			 notReliable:=TRUE;
  		    END_IF;
  		ELSE
  		    IF (ABS(strAI.ChangeSpeed)>strAI.maxChangeSpeedDown) AND (strAI.maxChangeSpeedDown>0.0000001)  THEN
                                 notReliable:=TRUE;
  		    END_IF;
  		END_IF;

  END_IF;

  strAI.status := SHL(BYTE_TO_DWORD(source_for_Status), 29) 		              (* Источник команды *)
  			OR SHL(BYTE_TO_DWORD(cmd_for_Status), 26) 	    (* Команда *)
  			OR SHL(BYTE_TO_DWORD(command_error_for_Status), 23)   (* Ошибка команды *)
  			OR SHL(BOOL_TO_DWORD(strAI.OpcCommandsDisabled ), 21) (* Управление в ВУ заблокировано *)
  			OR SHL(BOOL_TO_DWORD(strAI.Disabled_HA), 9)		    (* ВА исключена из формирования интервала *)
  			OR SHL(BOOL_TO_DWORD(strAI.Disabled_LA), 8)		    (* НА исключена из формирования интервала *)
  			OR SHL(BOOL_TO_DWORD(strAI.Disabled_HW), 7)		    (* ВП исключена из формирования интервала *)
  			OR SHL(BOOL_TO_DWORD(strAI.Disabled_LW), 6)	              (* НП исключена из формирования интервала *)
  			OR SHL(BOOL_TO_DWORD(strAI.NS), 5)			    (* неиспарвность сигнала *)
  			OR SHL(BOOL_TO_DWORD(strAI.remont), 4)	              (* Выведен в ремонт *)
  			OR BYTE_TO_DWORD(strAI.interval);	              (* интервал *)
END_FUNCTION_BLOCK

FUNCTION_BLOCK fb_AiProtection_Init
  VAR_INPUT
    data_Ini : BOOL;
    controlLimit : BYTE;
    delay : TIME;
    inTag : BYTE;
    inRunOnStart : BOOL;
  END_VAR
  VAR_IN_OUT
    str_AIp : struct_AiProtection;
  END_VAR
  VAR_OUTPUT
    Init : BOOL          := FALSE;
  END_VAR

  (*****            Функциональный блок переинициализации структуры  AiProtection          *****)

   Init := FALSE;

      IF data_Ini THEN                            (* Параметрам требуется переинициализация. *)
          str_AIp.controlLimit        := controlLimit;
          str_AIp.delay               := delay;
          str_AIp.inTag               := inTag;
          str_AIp.inRunOnStart        := inRunOnStart;

          data_Ini:=FALSE;
          Init := TRUE;
      END_IF;
      IF Init THEN
          controlLimit:= 0;
          delay:= T#0S;
          inTag:= 0;
          inRunOnStart:= FALSE;
      END_IF;
END_FUNCTION_BLOCK

FUNCTION_BLOCK proc_AI_Init
  VAR_INPUT
    init : BOOL;
  END_VAR
  VAR
    stAI_Ini : fb_AI_Init;
    inits : UINT;
  END_VAR
  VAR_INPUT
    initiales : UINT;
  END_VAR
  VAR_EXTERNAL
    ai : AiConfig;
  END_VAR

  inits := 0; (* Флаг необходимости инициализации структур-дескрипторов *)

  (********************************************* Модуль A2-14 ******************************************************)
  (* [A2-14, AI0-0] TStalisStatoraKanal1 *)
  stAI_Ini(data_Ini := TRUE, dLL := 0.0, dHL := 150.0,
  ISVALIDREF_HW := TRUE, dHW := 130.0, aperturFilter:= 0.5,
  strAI := ai.Tstali_statora_kanal_1);
  inits := inits + BOOL_TO_UINT(stAI_Ini.Init);

  (* [A2-14, AI0-1] TStalisStatoraKanal2 *)
  stAI_Ini(data_Ini := TRUE,  dLL := 0.0, dHL := 150.0,
  ISVALIDREF_HW := TRUE, dHW := 130.0, aperturFilter:= 0.5,
  strAI := ai.Tstali_statora_kanal_2);
  inits := inits + BOOL_TO_UINT(stAI_Ini.Init);

  (* [A2-14, AI0-2] TStalisStatoraKanal3 *)
  stAI_Ini(data_Ini := TRUE,  dLL := 0.0, dHL :=150.0,
  ISVALIDREF_HW := TRUE, dHW := 130.0, aperturFilter:= 0.5,
  strAI := ai.Tstali_statora_kanal_3);
  inits := inits + BOOL_TO_UINT(stAI_Ini.Init);

  (* [A2-14, AI0-3] TMediStatoraKanal1 *)
  stAI_Ini(data_Ini := TRUE,  dLL := 0.0, dHL := 150.0,
  ISVALIDREF_HW := TRUE, dHW := 130.0, aperturFilter:= 0.5,
  strAI := ai.Tmedi_statora_kanal_1);
  inits := inits + BOOL_TO_UINT(stAI_Ini.Init);

  (********************************************* Модуль A2-15 ******************************************************)

  (* [A2-15, AI1-0] TMediStatoraKanal2 *)
  stAI_Ini(data_Ini :=TRUE,  dLL := 0.0, dHL := 150.0,
  ISVALIDREF_HW := TRUE, dHW := 130.0, aperturFilter:= 0.5,
  strAI := ai.Tmedi_statora_kanal_2);
  inits := inits + BOOL_TO_UINT(stAI_Ini.Init);

  (* [A2-15, AI1-1] TMediStatoraKanal3 *)
  stAI_Ini(data_Ini := TRUE,  dLL := 0.0, dHL := 150.0,
  ISVALIDREF_HW := TRUE, dHW := 130.0, aperturFilter:= 0.5,
  strAI := ai.Tmedi_statora_kanal_3);
  inits := inits + BOOL_TO_UINT(stAI_Ini.Init);

  (* [A2-15, AI1-2] TOpornogoPodshipnikaEDT_1 *)
  stAI_Ini(data_Ini := TRUE,  dLL := 0.0, dHL := 100.0,
  ISVALIDREF_HA := TRUE, ISVALIDREF_HW := TRUE, dHA := 80.0, dHW := 75.0, aperturFilter:= 0.5, dMaxChangeSpeed := 10.0,
  strAI := ai.Toporno_podshipnika_EDT_1);
  inits := inits + BOOL_TO_UINT(stAI_Ini.Init);

  (* [A2-15, AI1-3]  TOpornoYpornogoPodshipnikaEDT_2 *)
  stAI_Ini(data_Ini := TRUE,  dLL := 0.0, dHL := 100.0,
  ISVALIDREF_HA := TRUE, ISVALIDREF_HW := TRUE, dHA := 80.0, dHW := 75.0, aperturFilter:= 0.5, dMaxChangeSpeed := 10.0,
  strAI := ai.Toy_podshipnika_EDT_2);
  inits := inits + BOOL_TO_UINT(stAI_Ini.Init);

  (********************************************* Модуль A3-1 ******************************************************)

  (* [A3-1, AI2-0]  TOpornoYpornogoPodshipnikaKolesaRedEDT_3 *)
  stAI_Ini(data_Ini := TRUE,  dLL := 0.0, dHL := 100.0,
  ISVALIDREF_HA := TRUE, ISVALIDREF_HW := TRUE, dHA := 80.0, dHW := 75.0, aperturFilter:= 0.5, dMaxChangeSpeed := 10.0,
  strAI := ai.Toy_podshipnika_kol_EDT_3);
  inits := inits + BOOL_TO_UINT(stAI_Ini.Init);

  (* [A3-1, AI2-1] TOpornoYpornogoPodshipnikaKolesaRedHT_4 *)
  stAI_Ini(data_Ini := TRUE,  dLL := 0.0, dHL := 100.0,
  ISVALIDREF_HA := TRUE, ISVALIDREF_HW := TRUE, dHA := 80.0, dHW := 75.0, aperturFilter:= 0.5, dMaxChangeSpeed := 10.0,
  strAI := ai.Toy_podshipnika_kol_EDT_4);
  inits := inits + BOOL_TO_UINT(stAI_Ini.Init);

  (* [A3-1, AI2-2] TOpornogoPodshipnikaShesterniReduktoraT_5 *)
  stAI_Ini(data_Ini := TRUE,  dLL := 0.0, dHL := 100.0,
  ISVALIDREF_HA := TRUE, ISVALIDREF_HW := TRUE, dHA := 80.0, dHW := 75.0, aperturFilter:= 0.5, dMaxChangeSpeed := 10.0,
  strAI := ai.Toy_podshipnika_shest_red_EDT_5);
  inits := inits + BOOL_TO_UINT(stAI_Ini.Init);

  (* [A3-1, AI2-3] TOpornogoPodshipnikaReduktoraHT_6 *)
  stAI_Ini(data_Ini := TRUE,  dLL := 0.0, dHL := 100.0,
  ISVALIDREF_HA := TRUE, ISVALIDREF_HW := TRUE, dHA := 80.0, dHW := 75.0, aperturFilter:= 0.5, dMaxChangeSpeed := 10.0,
  strAI := ai.Ty_podshipnika_red_EDT_6);
  inits := inits + BOOL_TO_UINT(stAI_Ini.Init);

  (********************************************* Модуль A3-2 ******************************************************)

  (* [A3-2, AI3-01]  TOpornoYpornogoPodshipnikaNagnetateljaT_7_1 *)
  stAI_Ini(data_Ini := TRUE,  dLL := 0.0, dHL := 100.0,
  ISVALIDREF_HA := TRUE, ISVALIDREF_HW := TRUE, dHA := 80.0, dHW := 75.0, aperturFilter:= 0.5, dMaxChangeSpeed := 10.0,
  strAI := ai.Ty_podshipnika_nagnet_EDT_7_1);
  inits := inits + BOOL_TO_UINT(stAI_Ini.Init);

  (* [A3-2, AI3-01]  TOpornoYpornogoPodshipnikaNagnetateljaT_7_2 *)
  stAI_Ini(data_Ini := TRUE,  dLL := 0.0, dHL := 100.0,
  ISVALIDREF_HA := TRUE, ISVALIDREF_HW := TRUE, dHA := 80.0, dHW := 75.0, aperturFilter:= 0.5, dMaxChangeSpeed := 10.0,
  strAI := ai.Ty_podshipnika_nagnet_EDT_7_2);
  inits := inits + BOOL_TO_UINT(stAI_Ini.Init);

  (* [A3-2, AI3-2]  TOpornoYpornogoPodshipnikaSvobodnogoKoncaNT_8_1 *)
  stAI_Ini(data_Ini := TRUE,  dLL := 0.0, dHL := 100.0,
  ISVALIDREF_HA := TRUE, ISVALIDREF_HW := TRUE, dHA := 80.0, dHW := 75.0, aperturFilter:= 0.5, dMaxChangeSpeed := 10.0,
  strAI := ai.Toy_podshipnika_svobod_konca_EDT_8_1);
  inits := inits + BOOL_TO_UINT(stAI_Ini.Init);

  (* [A3-2, AI3-2]  TOpornoYpornogoPodshipnikaSvobodnogoKoncaNT_8_2 *)
  stAI_Ini(data_Ini := TRUE,  dLL := 0.0, dHL := 100.0,
  ISVALIDREF_HA := TRUE, ISVALIDREF_HW := TRUE, dHA := 80.0, dHW := 75.0, aperturFilter:= 0.5, dMaxChangeSpeed := 10.0,
  strAI := ai.Toy_podshipnika_svobod_konca_EDT_8_2);
  inits := inits + BOOL_TO_UINT(stAI_Ini.Init);

  (********************************************* Модуль A3-3 ******************************************************)

  (* [A3-3, AI4-1]  TYpornogoPodshipnikaRavKolodokHT_9_1 *)
  stAI_Ini(data_Ini := TRUE,  dLL := 0.0, dHL := 100.0,
  ISVALIDREF_HA := TRUE, ISVALIDREF_HW := TRUE, dHA := 80.0, dHW := 75.0, aperturFilter:= 0.5, dMaxChangeSpeed := 10.0,
  strAI := ai.Toy_podshipnika_rab_kol_EDT_9_1);
  inits := inits + BOOL_TO_UINT(stAI_Ini.Init);

  (* [A3-3, AI4-1]  TYpornogoPodshipnikaRavKolodokHT_9_2 *)
  stAI_Ini(data_Ini := TRUE,  dLL := 0.0, dHL := 100.0,
  ISVALIDREF_HA := TRUE, ISVALIDREF_HW := TRUE, dHA := 80.0, dHW := 75.0, aperturFilter:= 0.5, dMaxChangeSpeed := 10.0,
  strAI := ai.Toy_podshipnika_rab_kol_EDT_9_2);
  inits := inits + BOOL_TO_UINT(stAI_Ini.Init);

  (* [A3-3, AI4-3] TYpornogoPodshipnikaNerabKolodokHT_10_1 *)
  stAI_Ini(data_Ini := TRUE,  dLL := 0.0, dHL := 100.0,
  ISVALIDREF_HA := TRUE, ISVALIDREF_HW := TRUE, dHA := 80.0, dHW := 75.0, aperturFilter:= 0.5, dMaxChangeSpeed := 10.0,
  strAI := ai.Toy_podshipnika_nerab_kol_EDT_10_1);
  inits := inits + BOOL_TO_UINT(stAI_Ini.Init);

  (* [A3-3, AI4-3] TYpornogoPodshipnikaNerabKolodokHT_10_2 *)
  stAI_Ini(data_Ini := TRUE,  dLL := 0.0, dHL := 100.0,
  ISVALIDREF_HA := TRUE, ISVALIDREF_HW := TRUE, dHA := 80.0, dHW := 75.0, aperturFilter:= 0.5, dMaxChangeSpeed := 10.0,
  strAI := ai.Toy_podshipnika_nerab_kol_EDT_10_2);
  inits := inits + BOOL_TO_UINT(stAI_Ini.Init);

  (********************************************* Модуль A3-4 ******************************************************)
  (* [A3-4, AI5-0] THolodnogoVozduhaEDKanall *)
  stAI_Ini(data_Ini := TRUE,  dLL := 0.0, dHL := 100.0,
  ISVALIDREF_HW := TRUE, dHW := 60.0, aperturFilter:= 0.5,
  strAI := ai.Tholodnogo_vozduha_ED_kanal_1);
  inits := inits + BOOL_TO_UINT(stAI_Ini.Init);

  (* [A3-4, AI5-1] THolodnogoVozduhaEDKanal2 *)
  stAI_Ini(data_Ini := TRUE,  dLL := 0.0, dHL := 100.0,
  ISVALIDREF_HW := TRUE, dHW := 60.0, aperturFilter:= 0.5,
  strAI := ai.Tholodnogo_vozduha_ED_kanal_2);
  inits := inits + BOOL_TO_UINT(stAI_Ini.Init);

  (* [A3-4, AI5-2]  TGorjachegoVozduhaEDKanall *)
  stAI_Ini(data_Ini := TRUE,  dLL := 0.0, dHL := 100.0,
  ISVALIDREF_HW := TRUE, dHW := 70.0, aperturFilter:= 0.5,
  strAI := ai.Tgorjachego_vozduha_ED_kanal_1);
  inits := inits + BOOL_TO_UINT(stAI_Ini.Init);

  (* [A3-4, AI5-3] TGorjachegoVozduhaEDKanal2 *)
  stAI_Ini(data_Ini := TRUE,  dLL := 0.0, dHL := 100.0,
  ISVALIDREF_HW := TRUE, dHW := 70.0, aperturFilter:= 0.5,
  strAI := ai.Tgorjachego_vozduha_ED_kanal_2);
  inits := inits + BOOL_TO_UINT(stAI_Ini.Init);

  (********************************************* Модуль A3-5 ******************************************************)

  (* [A3-5, AI6-0] TNArujnogoVozduha *)
  stAI_Ini(data_Ini := TRUE,  dLL := -50.0, dHL := 100.0,
  ISVALIDREF_HW := TRUE, dHW := 70.0, aperturFilter:= 0.5,
  strAI := ai.Tnarujnogo_vozduha);
  inits := inits + BOOL_TO_UINT(stAI_Ini.Init);

  (* [A3-5, AI6-1]  TgazaNaVhodeH *)
  stAI_Ini(data_Ini := TRUE,  dLL := -50.0, dHL := 100.0,
  ISVALIDREF_HW := TRUE, dHW := 80.0, aperturFilter:= 0.5,
  strAI := ai.Tgaza_na_vhode_H);
  inits := inits + BOOL_TO_UINT(stAI_Ini.Init);

  (* [A3-5, AI6-2] TgazaNaVyhodeH *)
  stAI_Ini(data_Ini := TRUE,  dLL := -50.0, dHL := 100.0,
  ISVALIDREF_HW := TRUE, ISVALIDREF_HA := TRUE, dHa :=90.0, dHW := 80.0, aperturFilter:= 0.5, dMaxChangeSpeed := 10.0,
  strAI := ai.Tgaza_na_vyhode_H);
  inits := inits + BOOL_TO_UINT(stAI_Ini.Init);

  (********************************************* Модуль A3-6 ******************************************************)
  (* [A3-6, AI7-0] TMasladoAVOM *)
  stAI_Ini(data_Ini := TRUE,  dLL := 0.0, dHL := 150.0,
  ISVALIDREF_HW := TRUE, dHW := 55.0, aperturFilter:= 0.5,
  strAI := ai.Tmasla_do_AVOM);
  inits := inits + BOOL_TO_UINT(stAI_Ini.Init);

  (* [A3-6, AI7-1] TMaslaPosleAVOM *)
  stAI_Ini(data_Ini := TRUE,  dLL := 0.0, dHL := 150.0,
  ISVALIDREF_HW := TRUE, dHW := 55.0, aperturFilter:= 0.5, dMaxChangeSpeed := 10.0,
  strAI := ai.Tmasla_posle_AVOM);
  inits := inits + BOOL_TO_UINT(stAI_Ini.Init);
  (********************************************* Модуль A3-8 ******************************************************)
  (* [A3-8, AI9-0]  TMaslaMB *)
  stAI_Ini(data_Ini := TRUE,  dLL := 0.0, dHL := 150.0,
  ISVALIDREF_LW := TRUE, dLW := 25.0, aperturFilter:= 0.5, dMaxChangeSpeed := 10.0,
  strAI := ai.Tmasla_MB);
  inits := inits + BOOL_TO_UINT(stAI_Ini.Init);

  (* [A3-6, AI7-2] TMaslaMB_TEN *)
  stAI_Ini(data_Ini := TRUE,  dLL := 0.0, dHL := 100.0,
  ISVALIDREF_HW := TRUE, dHW := 50.0, aperturFilter:= 0.5, dMaxChangeSpeed := 10.0,
  strAI := ai.Tmasla_MB_TEN);
  inits := inits + BOOL_TO_UINT(stAI_Ini.Init);

  (* [A3-8, AI9-1]  TEmperatura_v_SHU *)
  stAI_Ini(data_Ini := TRUE,  dLL := -40.0, dHL := 100.0, CurrentShotCircuit := 20320.0, CurrentBreakCircuit := 3680.0,
  aperturFilter:= 0.5, strAI := ai.Tshu);
  inits := inits + BOOL_TO_UINT(stAI_Ini.Init);

  (* [A3-8, AI9-2]  DavlenijaMasloSmNizkoe *)
  stAI_Ini(data_Ini := TRUE,  dLL := 0.0, dHL := 250.0,
  ISVALIDREF_LW := TRUE, ISVALIDREF_LA := TRUE, dLW := 50.0, dLA := 25.0,  CurrentShotCircuit := 20240.0, CurrentBreakCircuit := 3760.0,  aperturFilter:= 0.5,
  strAI := ai.Pmaslo_sm_nizkoe);
  inits := inits + BOOL_TO_UINT(stAI_Ini.Init);

  (* [A3-8, AI9-3]  PerepadDavlenieNaMasloFiltre *)
  stAI_Ini(data_Ini := TRUE,  dLL := 0.0, dHL := 250.0,
  ISVALIDREF_HW := TRUE, dHW := 150.0, CurrentShotCircuit := 20240.0, CurrentBreakCircuit := 3760.0, aperturFilter:= 0.5,
  strAI := ai.dPgaza_na_maslo_filtre);
  inits := inits + BOOL_TO_UINT(stAI_Ini.Init);

  (********************************************* Модуль A3-9 ******************************************************)
  (* [A3-9, AI10-0]  DavlenijaMasloSmVysokoe *)
  stAI_Ini(data_Ini := TRUE,  dLL := 0.0, dHL := 1000.0,
  ISVALIDREF_LW := TRUE, ISVALIDREF_LA := TRUE, dLW := 300.0, dLA := 250.0, CurrentShotCircuit := 20240.0, CurrentBreakCircuit := 3760.0, aperturFilter:= 0.5,
  strAI := ai.Pmaslo_sm_vysokoe);
  inits := inits + BOOL_TO_UINT(stAI_Ini.Init);

  (* [A3-9, AI10-1]  DavlenijaMaslaPosleGNS *)
  stAI_Ini(data_Ini := TRUE,  dLL := 0.0, dHL := 250.0, aperturFilter:= 0.5, CurrentShotCircuit := 20240.0, CurrentBreakCircuit := 3760.0,
  ISVALIDREF_LW := TRUE, ISVALIDREF_HW := TRUE,
  dLW := 187.0, dHW := 242.0,
  strAI := ai.Pmasla_posle_GNS);
  inits := inits + BOOL_TO_UINT(stAI_Ini.Init);

  (* [A3-9, AI10-2] DavlenijaMaslaPosleNU *)
  stAI_Ini(data_Ini := TRUE,  dLL := 0.0, dHL := 10.0, aperturFilter:= 0.5, CurrentShotCircuit := 20240.0, CurrentBreakCircuit := 3760.0,
  ISVALIDREF_LW := TRUE, dLW := 3.0,
  strAI := ai.Pmasla_posle_NU);
  inits := inits + BOOL_TO_UINT(stAI_Ini.Init);

  (********************************************* Модуль A3-10 ******************************************************)
  (* [A3-10, AI11-0] PerepadDavlenieNaKonfuzore *)
  stAI_Ini(data_Ini := TRUE,  dLL := 0.0, dHL := 250.0,
  ISVALIDREF_LW := TRUE, dLW := 15.0, aperturFilter:= 0.5, CurrentShotCircuit := 20240.0, CurrentBreakCircuit := 3760.0,
  strAI := ai.dPgaza_na_konfuzore);
  inits := inits + BOOL_TO_UINT(stAI_Ini.Init);

  (* [A3-10, AI11-1] OsSdvigNagnetatelja_Plus *)
  stAI_Ini(data_Ini := TRUE,  dLL := 0.0, dHL := 1000.0,
  ISVALIDREF_HA := TRUE, ISVALIDREF_HW := TRUE, dHW := 200.0, dHA := 300.0, aperturFilter := 0.5, CurrentShotCircuit := 20240.0, CurrentBreakCircuit := 3760.0,
  strAI := ai.Os_sdvig_nagnetatelja_plus);
  inits := inits + BOOL_TO_UINT(stAI_Ini.Init);

  (* [A3-10, AI11-2] OsSdvigNagnetatelja_Minus *)
  stAI_Ini(data_Ini := TRUE,  dLL := 0.0, dHL := 1600.0,
  ISVALIDREF_LW := TRUE, dLW := 150.0, ISVALIDREF_LA := TRUE, dLA := 100.0, aperturFilter := 0.5, CurrentShotCircuit := 20240.0, CurrentBreakCircuit := 3760.0,
  strAI := ai.Os_sdvig_nagnetatelja_minus);
  inits := inits + BOOL_TO_UINT(stAI_Ini.Init);

  (* [A3-10, AI11-3] PerepadDavlenieMasloGaz *)
  stAI_Ini(data_Ini := TRUE, dLL := 0.0, dHL := 1600.0,
  ISVALIDREF_LW := TRUE, ISVALIDREF_LA := TRUE, dLW := 150.0, dLa := 100.0, aperturFilter:= 0.5, CurrentShotCircuit := 20240.0, CurrentBreakCircuit := 3760.0,
  strAI := ai.dPmaslo_gaz);
  inits := inits + BOOL_TO_UINT(stAI_Ini.Init);

  (********************************************* Модуль A3-11 ******************************************************)
  (* [A3-11, AI12-0]  DGazaNaVhodeNagnetatelja *)
  stAI_Ini(data_Ini := TRUE,  dLL := 0.0, dHL := 10.0,
  ISVALIDREF_LW := TRUE, dLW := 4.895, aperturFilter := 0.5, CurrentShotCircuit := 20240.0, CurrentBreakCircuit := 3760.0,
  strAI := ai.Pgaza_na_vhode_nagnetatelia);
  inits := inits + BOOL_TO_UINT(stAI_Ini.Init);

  (* [A3-11, AI12-1]  DGazaNaVyhodeNagnetatelja *)
  stAI_Ini(data_Ini := TRUE,  dLL := 0.0, dHL := 10.0,
  ISVALIDREF_HA := TRUE, ISVALIDREF_HW := TRUE, dLA := 7.653, dHW := 7.55, aperturFilter := 0.5, CurrentShotCircuit := 20240.0, CurrentBreakCircuit := 3760.0,
  strAI := ai.Pgaza_na_vyhode_nagnetatelia);
  inits := inits + BOOL_TO_UINT(stAI_Ini.Init);

  (* [A3-11, AI12-3]  DavlenieImpulsGaz *)
  stAI_Ini(data_Ini := TRUE,  dLL := 0.0, dHL := 10.0,
  ISVALIDREF_LW := TRUE, dLW := 5.0, aperturFilter := 0.5, CurrentShotCircuit := 20240.0, CurrentBreakCircuit := 3760.0,
  strAI := ai.Pimpuls_gaz);
  inits := inits + BOOL_TO_UINT(stAI_Ini.Init);

  (********************************************* Модуль A3-12 ******************************************************)
  (* [A3-12, AI13-0] YrovenMaslaMB *)
  stAI_Ini(data_Ini := TRUE,  dLL := 190.0, dHL := 885.0,
  ISVALIDREF_LW := TRUE, dLW := 530.0, aperturFilter := 0.5,  CurrentShotCircuit := 20240.0, CurrentBreakCircuit := 3760.0,
  strAI := ai.Yroven_masla_MB);
  inits := inits + BOOL_TO_UINT(stAI_Ini.Init);

  (********************************************* Модуль A3-13 ******************************************************)
  (* [A3-13, AI14-0]  Kontrol_per220V *)
  stAI_Ini(data_Ini := TRUE,  dLL := 0.0, dHL := 250.0,
  ISVALIDREF_LW := TRUE, ISVALIDREF_HW := TRUE, dLW := 187.0, dHW := 242.0, aperturFilter := 0.5, CurrentShotCircuit := 20240.0, CurrentBreakCircuit := 3760.0,
  strAI := ai.Kontrol_per_220V);
  inits := inits + BOOL_TO_UINT(stAI_Ini.Init);

  (* [A3-13, AI14-1]  Kontrol_post220V *)
  stAI_Ini(data_Ini := TRUE,  dLL := 0.0, dHL := 250.0,
  ISVALIDREF_HW := TRUE, ISVALIDREF_LW := TRUE, dHW := 242.0, dLW := 187.0, aperturFilter := 0.5, CurrentShotCircuit := 20240.0, CurrentBreakCircuit := 3760.0,
  strAI := ai.Kontrol_post_220V);
  inits := inits + BOOL_TO_UINT(stAI_Ini.Init);

  (* [A3-13, AI14-2]  VibroSkorostOPED_T1 *)
  stAI_Ini(data_Ini := TRUE,  dLL := 0.0, dHL := 25.0,
  ISVALIDREF_HW := TRUE, ISVALIDREF_HA := TRUE, dHW := 11.0, dHA := 18.0, aperturFilter := 0.5, CurrentShotCircuit := 20240.0, CurrentBreakCircuit := 3760.0,
  strAI := ai.Vibro_skorost_OPED_T1);
  inits := inits + BOOL_TO_UINT(stAI_Ini.Init);

  (* [A3-13, AI14-3]  VibroSkorostOYPED_T2 *)
  stAI_Ini(data_Ini := TRUE,  dLL := 0.0, dHL := 25.0,
  ISVALIDREF_HW := TRUE, ISVALIDREF_HA := TRUE, dHW := 11.0, dHA := 18.0, aperturFilter := 0.5, CurrentShotCircuit := 20240.0, CurrentBreakCircuit := 3760.0,
  strAI := ai.Vibro_skorost_OYPED_T2);
  inits := inits + BOOL_TO_UINT(stAI_Ini.Init);

  (********************************************* Модуль A3-14 ******************************************************)
  (* [A3-14, AI15-0]  VibroSkorostOYPKolesaED_T3 *)
  stAI_Ini(data_Ini := TRUE,  dLL := 0.0, dHL := 25.0,
  ISVALIDREF_HW := TRUE, ISVALIDREF_HA := TRUE, dHW := 11.0, dHA := 18.0, aperturFilter := 0.5, CurrentShotCircuit := 20240.0, CurrentBreakCircuit := 3760.0,
  strAI := ai.Vibro_skorost_OYP_kolesa_ED_T3);
  inits := inits + BOOL_TO_UINT(stAI_Ini.Init);

  (* [A3-14, AI15-1]  VibroSkorostOPKolesaRH_T4 *)
  stAI_Ini(data_Ini := TRUE,  dLL := 0.0, dHL := 25.0,
  ISVALIDREF_HW := TRUE, ISVALIDREF_HA := TRUE, dHW := 11.0, dHA := 18.0, aperturFilter := 0.5, CurrentShotCircuit := 20240.0, CurrentBreakCircuit := 3760.0,
  strAI := ai.Vibro_skorost_OP_kolesa_RH_T4);
  inits := inits + BOOL_TO_UINT(stAI_Ini.Init);

  (* [A3-11, AI12-2]  VibroSkorostOPShesterniRED_T5 *)
  stAI_Ini(data_Ini := TRUE,  dLL := 0.0, dHL := 25.0,
  ISVALIDREF_HW := TRUE, ISVALIDREF_HA := TRUE, dHW := 11.0, dHA := 18.0, aperturFilter := 0.5, CurrentShotCircuit := 20240.0, CurrentBreakCircuit := 3760.0,
  strAI := ai.Vibro_skorost_OP_shesterni_RED_T5);
  inits := inits + BOOL_TO_UINT(stAI_Ini.Init);

  (* [A3-11, AI12-2]  VibroSkorostOPShesterniRED_T5 *)
  stAI_Ini(data_Ini := TRUE,  dLL := 0.0, dHL := 25.0,
  ISVALIDREF_HW := TRUE, ISVALIDREF_HA := TRUE, dHW := 11.0, dHA := 18.0, aperturFilter := 0.5, CurrentShotCircuit := 20240.0, CurrentBreakCircuit := 3760.0,
  strAI := ai.Vibro_skorost_OP_shesterni_RED_T6);
  inits := inits + BOOL_TO_UINT(stAI_Ini.Init);

  (* [A3-11, AI12-2]  VibroSkorostOPShesterniRED_T5 *)
  stAI_Ini(data_Ini := TRUE,  dLL := 0.0, dHL := 1000.0,
  ISVALIDREF_LW := TRUE, dLW := 300.0, aperturFilter := 0.5, CurrentShotCircuit := 20240.0, CurrentBreakCircuit := 3760.0,
  strAI := ai.Tok_statora);
  inits := inits + BOOL_TO_UINT(stAI_Ini.Init);

  initiales := 0;
  IF init THEN initiales := inits; END_IF;
END_FUNCTION_BLOCK

FUNCTION_BLOCK proc_AI
  VAR
    fb_TStalisStatoraKanal1 : fb_AiSourceMlp;
    fb_TStalisStatoraKanal2 : fb_AiSourceMlp;
    fb_TStalisStatoraKanal3 : fb_AiSourceMlp;
    fb_TMediStatoraKanal1 : fb_AiSourceMlp;
    fb_TMediStatoraKanal2 : fb_AiSourceMlp;
    fb_TMediStatoraKanal3 : fb_AiSourceMlp;
    fb_TOpornogoPodshipnikaEDT_1 : fb_AiSourceMlp;
    fb_TOpornoYpornogoPodshipnikaEDT_2 : fb_AiSourceMlp;
    fb_TOpornoYpornogoPodshipnikaKolesaRedEDT_3 : fb_AiSourceMlp;
    fb_TOpornoYpornogoPodshipnikaKolesaRedHT_4 : fb_AiSourceMlp;
    fb_TOpornogoPodshipnikaShesterniReduktoraT_5 : fb_AiSourceMlp;
    fb_TOpornogoPodshipnikaReduktoraHT_6 : fb_AiSourceMlp;
    fb_TOpornoYpornogoPodshipnikaNagnetateljaT_7_1 : fb_AiSourceMlp;
    fb_TOpornoYpornogoPodshipnikaNagnetateljaT_7_2 : fb_AiSourceMlp;
    fb_TOpornoYpornogoPodshipnikaSvobodnogoKoncaNT_8_1 : fb_AiSourceMlp;
    fb_TOpornoYpornogoPodshipnikaSvobodnogoKoncaNT_8_2 : fb_AiSourceMlp;
    fb_TYpornogoPodshipnikaRabKolodokHT_9_1 : fb_AiSourceMlp;
    fb_TYpornogoPodshipnikaRabKolodokHT_9_2 : fb_AiSourceMlp;
    fb_TYpornogoPodshipnikYstanKolodokHT_10_1 : fb_AiSourceMlp;
    fb_TYpornogoPodshipnikYstanKolodokHT_10_2 : fb_AiSourceMlp;
    fb_THolodnogoVozduhaEDKanall : fb_AiSourceMlp;
    fb_THolodnogoVozduhaEDKanal2 : fb_AiSourceMlp;
    fb_TGorjachegoVozduhaEDKanall : fb_AiSourceMlp;
    fb_TGorjachegoVozduhaEDKanal2 : fb_AiSourceMlp;
    fb_TNArujnogoVozduha : fb_AiSourceMlp;
    fb_TgazaNaVhodeH : fb_AiSourceMlp_timer;
    fb_TgazaNaVyhodeH : fb_AiSourceMlp;
    fb_TMasladoAVOM : fb_AiSourceMlp;
    fb_TMaslaPosleAVOM : fb_AiSourceMlp;
    fb_TMaslaMB : fb_AiSourceMlp;
    fb_TEmperatura_v_SHU : fb_AiSourceMlp_timer;
    fb_DavlenijaMasloSmNizkoe : fb_AiSourceMlp;
    fb_PerepadDavlenieNaMasloFiltre : fb_AiSourceMlp;
    fb_DavlenijaMasloSmVysokoe : fb_AiSourceMlp;
    fb_DavlenijaMaslaPosleGNS : fb_AiSourceMlp;
    fb_DavlenijaMaslaPosleNU : fb_AiSourceMlp;
    fb_PerepadDavlenieNaKonfuzore : fb_AiSourceMlp;
    fb_OsSdvigNagnetatelja_Plus : fb_AiSourceMlp;
    fb_OsSdvigNagnetatelja_Minus : fb_AiSourceMlp;
    fb_PerepadDavlenieMasloGaz : fb_AiSourceMlp;
    fb_VibroSkorostOYPKolesaED_T3 : fb_AiSourceMlp;
    fb_DGazaNaVhodeNagnetatelja : fb_AiSourceMlp;
    fb_DGazaNaVyhodeNagnetatelja : fb_AiSourceMlp;
    fb_DavlenieImpulsGaz : fb_AiSourceMlp;
    fb_YrovenMaslaMB : fb_AiSourceMlp;
    fb_Kontrol_per220V : fb_AiSourceMlp;
    fb_Kontrol_post220V : fb_AiSourceMlp;
    fb_TMaslaMB_TEN : fb_AiSourceMlp;
    fb_VibroSkorostOPED_T1 : fb_AiSourceMlp;
    fb_VibroSkorostOYPED_T2 : fb_AiSourceMlp;
    fb_VibroSkorostOPKolesaRH_T4 : fb_AiSourceMlp;
    fb_VibroSkorostOPShesterniRED_T5 : fb_AiSourceMlp;
    fb_VibroSkorostOPShesterniReduktoraH_T6 : fb_AiSourceMlp;
    fb_TokStatora : fb_AiSourceMlp;
  END_VAR
  VAR_EXTERNAL
    arAIN_0 : TItemAIN;
    arAIN_1 : TItemAIN;
    arAIN_2 : TItemAIN;
    arAIN_3 : TItemAIN;
    arAIN_4 : TItemAIN;
    arAIN_5 : TItemAIN;
    arAIN_6 : TItemAIN;
    arAIN_7 : TItemAIN;
    arAIN_8 : TItemAIN;
    arAIN_9 : TItemAIN;
    arAIN_10 : TItemAIN;
    arAIN_11 : TItemAIN;
    arAIN_12 : TItemAIN;
    arAIN_13 : TItemAIN;
    arAIN_14 : TItemAIN;
    arAIN_15 : TItemAIN;
    ai : AiConfig;
    arAIN_16 : TItemAIN;
    arAIN_17 : TItemAIN;
    arAIN_18 : TItemAIN;
    arAIN_19 : TItemAIN;
    arAIN_20 : TItemAIN;
    arAIN_21 : TItemAIN;
    arAIN_22 : TItemAIN;
    arAIN_23 : TItemAIN;
    arAIN_24 : TItemAIN;
    arAIN_25 : TItemAIN;
    arAIN_26 : TItemAIN;
    arAIN_27 : TItemAIN;
    arAIN_28 : TItemAIN;
    arAIN_29 : TItemAIN;
    arAIN_30 : TItemAIN;
    arAIN_31 : TItemAIN;
    arAIN_32 : TItemAIN;
    arAIN_33 : TItemAIN;
    arAIN_34 : TItemAIN;
    arAIN_35 : TItemAIN;
    arAIN_36 : TItemAIN;
    arAIN_37 : TItemAIN;
    arAIN_38 : TItemAIN;
    arAIN_39 : TItemAIN;
    arAIN_40 : TItemAIN;
    arAIN_41 : TItemAIN;
    arAIN_42 : TItemAIN;
    arAIN_43 : TItemAIN;
    arAIN_44 : TItemAIN;
    arAIN_45 : TItemAIN;
    arAIN_46 : TItemAIN;
    arAIN_47 : TItemAIN;
    arAIN_48 : TItemAIN;
    arAIN_49 : TItemAIN;
    arAIN_50 : TItemAIN;
    arAIN_51 : TItemAIN;
    arAIN_52 : TItemAIN;
    arAIN_53 : TItemAIN;
    arAIN_54 : TItemAIN;
    arAIN_55 : TItemAIN;
    arAIN_56 : TItemAIN;
    arAIN_57 : TItemAIN;
    arAIN_58 : TItemAIN;
    arAIN_59 : TItemAIN;
    arAIN_60 : TItemAIN;
    arAIN_61 : TItemAIN;
    arAIN_62 : TItemAIN;
    arAIN_63 : TItemAIN;
    arAIN_64 : TItemAIN;
    arAIN_65 : TItemAIN;
    arERR_3 : TItemDIN;
    arERR_4 : TItemDIN;
    arERR_5 : TItemDIN;
    arERR_6 : TItemDIN;
    arERR_7 : TItemDIN;
    arERR_8 : TItemDIN;
    arERR_9 : TItemDIN;
    A1_10_err_mode : UINT;
    A1_11_err_mode : UINT;
    A1_4_err_mode : UINT;
    A1_5_err_mode : UINT;
    A1_6_err_mode : UINT;
    A1_7_err_mode : UINT;
    A1_8_err_mode : UINT;
    A1_9_err_mode : UINT;
    A2_2_err_mode : UINT;
    A2_3_err_mode : UINT;
    AI_0_dblValue : LREAL;
    AI_10_dblValue : LREAL;
    AI_11_dblValue : LREAL;
    AI_12_dblValue : LREAL;
    AI_13_dblValue : LREAL;
    AI_14_dblValue : LREAL;
    AI_15_dblValue : LREAL;
    AI_16_dblValue : LREAL;
    AI_17_dblValue : LREAL;
    AI_18_dblValue : LREAL;
    AI_19_dblValue : LREAL;
    AI_1_dblValue : LREAL;
    AI_20_dblValue : LREAL;
    AI_21_dblValue : LREAL;
    AI_22_dblValue : LREAL;
    AI_23_dblValue : LREAL;
    AI_24_dblValue : LREAL;
    AI_25_dblValue : LREAL;
    AI_26_dblValue : LREAL;
    AI_27_dblValue : LREAL;
    AI_28_dblValue : LREAL;
    AI_29_dblValue : LREAL;
    AI_2_dblValue : LREAL;
    AI_30_dblValue : LREAL;
    AI_31_dblValue : LREAL;
    AI_32_dblValue : LREAL;
    AI_33_dblValue : LREAL;
    AI_34_dblValue : LREAL;
    AI_35_dblValue : LREAL;
    AI_36_dblValue : LREAL;
    AI_37_dblValue : LREAL;
    AI_38_dblValue : LREAL;
    AI_39_dblValue : LREAL;
    AI_3_dblValue : LREAL;
    AI_40_dblValue : LREAL;
    AI_41_dblValue : LREAL;
    AI_42_dblValue : LREAL;
    AI_43_dblValue : LREAL;
    AI_44_dblValue : LREAL;
    AI_45_dblValue : LREAL;
    AI_46_dblValue : LREAL;
    AI_47_dblValue : LREAL;
    AI_48_dblValue : LREAL;
    AI_49_dblValue : LREAL;
    AI_4_dblValue : LREAL;
    AI_50_dblValue : LREAL;
    AI_51_dblValue : LREAL;
    AI_52_dblValue : LREAL;
    AI_53_dblValue : LREAL;
    AI_54_dblValue : LREAL;
    AI_55_dblValue : LREAL;
    AI_56_dblValue : LREAL;
    AI_57_dblValue : LREAL;
    AI_58_dblValue : LREAL;
    AI_59_dblValue : LREAL;
    AI_5_dblValue : LREAL;
    AI_60_dblValue : LREAL;
    AI_61_dblValue : LREAL;
    AI_62_dblValue : LREAL;
    AI_63_dblValue : LREAL;
    AI_64_dblValue : LREAL;
    AI_65_dblValue : LREAL;
    AI_66_dblValue : LREAL;
    AI_67_dblValue : LREAL;
    AI_68_dblValue : LREAL;
    AI_69_dblValue : LREAL;
    AI_6_dblValue : LREAL;
    AI_70_dblValue : LREAL;
    AI_71_dblValue : LREAL;
    AI_72_dblValue : LREAL;
    AI_73_dblValue : LREAL;
    AI_74_dblValue : LREAL;
    AI_75_dblValue : LREAL;
    AI_76_dblValue : LREAL;
    AI_77_dblValue : LREAL;
    AI_78_dblValue : LREAL;
    AI_79_dblValue : LREAL;
    AI_7_dblValue : LREAL;
    AI_8_dblValue : LREAL;
    AI_9_dblValue : LREAL;
  END_VAR

  (* Циклический опрос. Входные аналоговые параметры *)

  (* [A1-9, AI5-4]  dР газа на конфузоре *)
  fb_PerepadDavlenieNaKonfuzore(arAIN := arAIN_40, strAI := ai.dPgaza_na_konfuzore, err_mod:=arERR_8);
  AI_40_dblValue := arAIN_40.dblValue;

  (* [A1-9, AI5-0] dР масла на масляном фильтре *)
  fb_PerepadDavlenieNaMasloFiltre(arAIN := arAIN_34, strAI := ai.dPgaza_na_maslo_filtre, err_mod:=arERR_8);
  AI_34_dblValue := arAIN_34.dblValue;

  (* [A1-9, AI5-7]  dР масло-газ *)
  fb_PerepadDavlenieMasloGaz(arAIN := arAIN_41, strAI := ai.dPmaslo_gaz, err_mod:=arERR_8);
  AI_41_dblValue := arAIN_41.dblValue;

  (* [A1-10, AI6-2] Р газа на входе нагнетателя *)
  fb_DGazaNaVhodeNagnetatelja(arAIN := arAIN_44, strAI := ai.Pgaza_na_vhode_nagnetatelia, err_mod:=arERR_9);
  AI_44_dblValue := arAIN_44.dblValue;

  (* [A1-10, AI6-3] Р газа на выходе нагнетателя *)
  fb_DGazaNaVyhodeNagnetatelja(arAIN := arAIN_45, strAI := ai.Pgaza_na_vyhode_nagnetatelia, err_mod:=arERR_9);
  AI_45_dblValue := arAIN_45.dblValue;

  (* [A1-9, AI5-3]  Р масла после НУ *)
  fb_DavlenijaMaslaPosleNU(arAIN := arAIN_37, strAI := ai.Pmasla_posle_NU, err_mod:=arERR_8);
  AI_37_dblValue := arAIN_37.dblValue;

  (* [A1-8, AI4-6]  Р масла смазки низкое) *)
  fb_DavlenijaMasloSmNizkoe(arAIN := arAIN_33, strAI := ai.Pmaslo_sm_nizkoe, err_mod:=arERR_7);
  AI_33_dblValue := arAIN_33.dblValue;

  (* [A1-9, AI5-2]  Р масла смазки после ГМНС *)
  fb_DavlenijaMaslaPosleGNS(arAIN := arAIN_36, strAI := ai.Pmasla_posle_GNS, err_mod:=arERR_8);
  AI_36_dblValue := arAIN_36.dblValue;

  (* [A1-9, AI5-1]  Р масла смазки высокое *)
  fb_DavlenijaMasloSmVysokoe(arAIN := arAIN_35, strAI := ai.Pmaslo_sm_vysokoe, err_mod:=arERR_8);
  AI_35_dblValue := arAIN_35.dblValue;

  (* [A1-7, AI3-2] Т наружного воздуха *)
  fb_TNArujnogoVozduha(arAIN := arAIN_24, strAI := ai.Tnarujnogo_vozduha, err_mod:=arERR_6);
  AI_24_dblValue := arAIN_24.dblValue;

  (* [A1-8, AI4-0]  Т газа на входе нагнетателя *)
  fb_TgazaNaVhodeH(arAIN := arAIN_25, strAI := ai.Tgaza_na_vhode_H, err_mod:=arERR_7);
  AI_25_dblValue := arAIN_25.dblValue;

  (* [A1-8, AI4-1] Т газа на выходе нагнетателя *)
  fb_TgazaNaVyhodeH(arAIN := arAIN_26, strAI := ai.Tgaza_na_vyhode_H, err_mod:=arERR_7);
  AI_26_dblValue := arAIN_26.dblValue;

  (* [A1-6, AI2-7]  Т горячего воздуха в ЭД, точка 1 *)
  fb_TGorjachegoVozduhaEDKanall(arAIN := arAIN_22, strAI := ai.Tgorjachego_vozduha_ED_kanal_1, err_mod:=arERR_5);
  AI_22_dblValue := arAIN_22.dblValue;

  (* [A1-7, AI3-0] Т горячего воздуха в ЭД, точка 2 *)
  fb_TGorjachegoVozduhaEDKanal2(arAIN := arAIN_23, strAI := ai.Tgorjachego_vozduha_ED_kanal_2, err_mod:=arERR_6);
  AI_23_dblValue := arAIN_23.dblValue;

  (* [A1-8, AI4-4] Т масла в маслобаке *)
  fb_TMaslaMB(arAIN := arAIN_29, strAI := ai.Tmasla_MB, err_mod:=arERR_7);
  AI_29_dblValue := arAIN_29.dblValue;

  (* [A1-8, AI4-4] Т масла в маслобаке над ТЭНом *)
  fb_TMaslaMB_TEN(arAIN := arAIN_30, strAI := ai.Tmasla_MB_TEN, err_mod:=arERR_7);
  AI_30_dblValue := arAIN_30.dblValue;

  (* [A1-8, AI4-2] Т масла до АВО М *)
  fb_TMasladoAVOM(arAIN := arAIN_27, strAI := ai.Tgorjachego_vozduha_ED_kanal_2, err_mod:=arERR_7);
  AI_27_dblValue := arAIN_27.dblValue;

  (* [A1-8, AI4-3] Т масла после АВО М *)
  fb_TMaslaPosleAVOM(arAIN := arAIN_28, strAI := ai.Tmasla_posle_AVOM, err_mod:=arERR_7);
  AI_28_dblValue := arAIN_28.dblValue;

  (* [A1-4, AI0-3] Т Т меди статора фаза 1 *)
  fb_TMediStatoraKanal1(arAIN := arAIN_3, strAI := ai.Tmedi_statora_kanal_1, err_mod:=arERR_3);
  AI_3_dblValue := arAIN_3.dblValue;

  (* [A1-4, AI0-4] Т обмотки фазы 3 канал *)
  fb_TMediStatoraKanal2(arAIN := arAIN_4, strAI := ai.Tmedi_statora_kanal_2, err_mod:=arERR_3);
  AI_4_dblValue := arAIN_4.dblValue;

  (* [A1-4, AI0-5] Т меди статора фаза 2 *)
  fb_TMediStatoraKanal3(arAIN := arAIN_5, strAI := ai.Tmedi_statora_kanal_3, err_mod:=arERR_3);
  AI_5_dblValue := arAIN_5.dblValue;

  (* [A1-4, AI0-6] Т ОП ЭД со стороны свободного конца (т.1) } *)
  fb_TOpornogoPodshipnikaEDT_1(arAIN := arAIN_6, strAI := ai.Toporno_podshipnika_EDT_1, err_mod:=arERR_3);
  AI_6_dblValue := arAIN_6.dblValue;

  (* [A1-5, AI1-0]  Т ОУП ЭД со стороны редуктора (т.2) *)
  fb_TOpornoYpornogoPodshipnikaEDT_2(arAIN := arAIN_7, strAI := ai.Toy_podshipnika_EDT_2, err_mod:=arERR_4);
  AI_7_dblValue := arAIN_7.dblValue;

  (* [A1-5, AI1-1]  Т ОУП колеса редуктора со стороны ЭД (т.3) *)
  fb_TOpornoYpornogoPodshipnikaKolesaRedEDT_3(arAIN := arAIN_8, strAI := ai.Toy_podshipnika_kol_EDT_3, err_mod:=arERR_4);
  AI_8_dblValue := arAIN_8.dblValue;

  (* [A1-5, AI1-2]Т ОП колеса редуктора со стороны Н (т.4) *)
  fb_TOpornoYpornogoPodshipnikaKolesaRedHT_4(arAIN := arAIN_9, strAI := ai.Toy_podshipnika_kol_EDT_4, err_mod:=arERR_4);
  AI_9_dblValue := arAIN_9.dblValue;

  (* [A1-5, AI1-3] Т ОП шестерни редуктора со стороны ЭД (т.5) *)
  fb_TOpornogoPodshipnikaShesterniReduktoraT_5(arAIN := arAIN_10, strAI := ai.Toy_podshipnika_shest_red_EDT_5, err_mod:=arERR_4);
  AI_10_dblValue := arAIN_10.dblValue;

  (* [A1-5, AI1-4]  Т ОП шестерни редуктора со стороны Н (т.6) *)
  fb_TOpornogoPodshipnikaReduktoraHT_6(arAIN := arAIN_11, strAI := ai.Ty_podshipnika_red_EDT_6, err_mod:=arERR_4);
  AI_11_dblValue := arAIN_11.dblValue;

  (* [A1-5, AI1-5]  Т ОП Н со стороны редуктора (т.7) *)
  fb_TOpornoYpornogoPodshipnikaNagnetateljaT_7_1(arAIN := arAIN_12, strAI := ai.Ty_podshipnika_nagnet_EDT_7_1, err_mod:=arERR_4);
  AI_12_dblValue := arAIN_12.dblValue;

  (* [A1-5, AI1-5]  Т ОП Н со стороны редуктора (т.7) *)
  fb_TOpornoYpornogoPodshipnikaNagnetateljaT_7_2(arAIN := arAIN_13, strAI := ai.Ty_podshipnika_nagnet_EDT_7_2, err_mod:=arERR_4);
  AI_13_dblValue := arAIN_13.dblValue;

  (* [A1-5, AI1-7]  Т ОП Н со стороны свободного вала (т.8) *)
  fb_TOpornoYpornogoPodshipnikaSvobodnogoKoncaNT_8_1(arAIN := arAIN_14, strAI := ai.Toy_podshipnika_svobod_konca_EDT_8_1, err_mod:=arERR_4);
  AI_14_dblValue := arAIN_14.dblValue;

  (* [A1-5, AI1-7]  Т ОП Н со стороны свободного вала (т.8) *)
  fb_TOpornoYpornogoPodshipnikaSvobodnogoKoncaNT_8_2(arAIN := arAIN_15, strAI := ai.Toy_podshipnika_svobod_konca_EDT_8_2, err_mod:=arERR_4);
  AI_15_dblValue := arAIN_15.dblValue;

  (* [A1-6, AI2-1]  Т УП рабочих колодок нагнетателя(т9) *)
  fb_TYpornogoPodshipnikaRabKolodokHT_9_1(arAIN := arAIN_16, strAI := ai.Toy_podshipnika_rab_kol_EDT_9_1, err_mod:=arERR_5);
  AI_16_dblValue := arAIN_16.dblValue;

  (* [A1-6, AI2-1]  Т УП рабочих колодок нагнетателя(т9) *)
  fb_TYpornogoPodshipnikaRabKolodokHT_9_2(arAIN := arAIN_17, strAI := ai.Toy_podshipnika_rab_kol_EDT_9_2, err_mod:=arERR_5);
  AI_17_dblValue := arAIN_17.dblValue;

  (* [A1-6, AI2-3]  Т ОП установочных колодок нагнетателя(т10) *)
  fb_TYpornogoPodshipnikYstanKolodokHT_10_1(arAIN := arAIN_18, strAI := ai.Toy_podshipnika_nerab_kol_EDT_10_1, err_mod:=arERR_5);
  AI_18_dblValue := arAIN_18.dblValue;

  (* [A1-6, AI2-3]  Т ОП установочных колодок нагнетателя(т10) *)
  fb_TYpornogoPodshipnikYstanKolodokHT_10_2(arAIN := arAIN_19, strAI := ai.Toy_podshipnika_nerab_kol_EDT_10_2, err_mod:=arERR_5);
  AI_19_dblValue := arAIN_19.dblValue;

  (* [A1-4, AI0-0] Т стали статора фаза 1 *)
  fb_TStalisStatoraKanal1(arAIN := arAIN_0, strAI := ai.Tstali_statora_kanal_1, err_mod:=arERR_3);
  AI_0_dblValue := arAIN_0.dblValue;

  (* [A1-4, AI0-1] Т стали статора фаза 2 *)
  fb_TStalisStatoraKanal2(arAIN := arAIN_1, strAI := ai.Tstali_statora_kanal_2, err_mod:=arERR_3);
  AI_1_dblValue := arAIN_1.dblValue;

  (* [A1-4, AI0-2] Т стали статора фаза 3 *)
  fb_TStalisStatoraKanal3(arAIN := arAIN_2, strAI := ai.Tstali_statora_kanal_3, err_mod:=arERR_3);
  AI_2_dblValue := arAIN_2.dblValue;

  (* [A1-6, AI2-5] Т холодного воздуха в ЭД, точка 1 *)
  fb_THolodnogoVozduhaEDKanall(arAIN := arAIN_20, strAI := ai.Tholodnogo_vozduha_ED_kanal_1, err_mod:=arERR_5);
  AI_20_dblValue := arAIN_20.dblValue;

  (* [A1-6, AI2-6] Т холодного воздуха в ЭД, точка 2 *)
  fb_THolodnogoVozduhaEDKanal2(arAIN := arAIN_21, strAI := ai.Tholodnogo_vozduha_ED_kanal_2, err_mod:=arERR_5);
  AI_21_dblValue := arAIN_21.dblValue;

  (* [A1-10, AI6-5] Уровень масла в маслобаке *)
  fb_YrovenMaslaMB(arAIN := arAIN_48, strAI := ai.Yroven_masla_MB, err_mod:=arERR_9);
  AI_48_dblValue := arAIN_48.dblValue;

  (* [A1-10, AI6-5] Уровень масла в маслобаке *)
  fb_VibroSkorostOPED_T1(arAIN := arAIN_56, strAI := ai.Kontrol_post_220V, err_mod:=arERR_9);
  AI_56_dblValue := arAIN_56.dblValue;

  (* [A1-10, AI6-5] Уровень масла в маслобаке *)
  fb_VibroSkorostOYPED_T2(arAIN := arAIN_57, strAI := ai.Vibro_skorost_OPED_T1, err_mod:=arERR_9);
  AI_57_dblValue := arAIN_57.dblValue;

  (* [A1-10, AI6-5] Уровень масла в маслобаке *)
  fb_VibroSkorostOPKolesaRH_T4(arAIN := arAIN_59, strAI := ai.Vibro_skorost_OP_kolesa_RH_T4, err_mod:=arERR_9);
  AI_59_dblValue := arAIN_59.dblValue;

  (* [A1-10, AI6-5] Уровень масла в маслобаке *)
  fb_VibroSkorostOPShesterniRED_T5(arAIN := arAIN_60, strAI := ai.Vibro_skorost_OP_shesterni_RED_T5, err_mod:=arERR_9);
  AI_60_dblValue := arAIN_60.dblValue;

  (* [A1-10, AI6-5] Уровень масла в маслобаке *)
  fb_VibroSkorostOPShesterniReduktoraH_T6(arAIN := arAIN_61, strAI := ai.Vibro_skorost_OP_shesterni_RED_T6, err_mod:=arERR_9);
  AI_61_dblValue := arAIN_61.dblValue;

  (**********************************************s Модуль A1-5 *********************************************************)
  A1_4_err_mode := arERR_3.wValue;
  A1_6_err_mode := arERR_5.wValue;
  A1_5_err_mode := arERR_4.wValue;
  A1_7_err_mode := arERR_6.wValue;

  (********************************************** Модуль A1-8 *********************************************************)
  (* [A1-8, AI4-5]  Температура в шкафу САУ *)
  fb_TEmperatura_v_SHU(arAIN := arAIN_32, strAI := ai.Tshu, err_mod:=arERR_7);
  AI_32_dblValue := arAIN_32.dblValue;

  (* [A1-9, AI5-5]  Вибрация ротора нагнетателя т.4 *)
  fb_OsSdvigNagnetatelja_Plus(arAIN := arAIN_42, strAI := ai.Os_sdvig_nagnetatelja_plus, err_mod:=arERR_8);
  AI_42_dblValue := arAIN_42.dblValue;

  (* [A1-9, AI5-6]  Осевой сдвиг ротора нагнетателя *)
  fb_OsSdvigNagnetatelja_Minus(arAIN := arAIN_43, strAI := ai.Os_sdvig_nagnetatelja_minus, err_mod:=arERR_8);
  AI_43_dblValue := arAIN_43.dblValue;

  A1_9_err_mode := arERR_8.wValue;

  (********************************************** Модуль A1-10 *********************************************************)
  (* [A1-10, AI6-0] Температура внутри шкафа *)
  fb_VibroSkorostOYPKolesaED_T3(arAIN := arAIN_58, strAI := ai.Vibro_skorost_OYP_kolesa_ED_T3, err_mod:=arERR_9);
  AI_58_dblValue := arAIN_58.dblValue;

  (* [A1-10, AI6-4] Активная мощность *)
  fb_DavlenieImpulsGaz(arAIN := arAIN_46, strAI := ai.Pimpuls_gaz, err_mod:=arERR_9);
  AI_46_dblValue := arAIN_46.dblValue;

  (* [A1-10, AI6-6]  Напряжение питания ШУ, основной ввод *)
  fb_Kontrol_per220V(arAIN := arAIN_52, strAI := ai.Kontrol_per_220V, err_mod:=arERR_9);
  AI_52_dblValue := arAIN_52.dblValue;

  (* [A1-10, AI6-7]  Напряжение питания ШУ, резервный ввод *)
  fb_Kontrol_post220V(arAIN := arAIN_53, strAI := ai.Kontrol_post_220V, err_mod:=arERR_9);
  AI_53_dblValue := arAIN_53.dblValue;

  (* [A1-10, AI6-7]  Напряжение питания ШУ, резервный ввод *)
  fb_TokStatora(arAIN := arAIN_65, strAI := ai.Tok_statora, err_mod:=arERR_9);
  AI_65_dblValue := arAIN_65.dblValue;

  A1_10_err_mode := arERR_9.wValue;
END_FUNCTION_BLOCK

FUNCTION anyProtectionSignaling : BOOL
  VAR_INPUT
    protections : ProtectionsConfig;
  END_VAR

  anyProtectionSignaling:=
  protections.Topornogo_podshipnika_EDT_1.Signaling OR
  protections.Toy_podshipnika_EDT_2.Signaling OR
  protections.Toy_podshipnika_kol_EDT_3.Signaling OR
  protections.Toy_podshipnika_kol_EDT_4.Signaling OR
  protections.To_podshipnika_shest_red_EDT_5.Signaling OR
  protections.To_podshipnika_shest_red_EDT_6.Signaling OR
  protections.To_podshipnika_N_EDT_7.Signaling OR
  protections.To_podshipnika_svob_konca_EDT_8.Signaling OR
  protections.Ty_podshipnika_rab_kol_EDT_9.Signaling OR
  protections.Typornogo_podshipnika_nerab_kolodok_HT_10.Signaling OR
  protections.Tgaza_na_vyhode_H.Signaling OR
  protections.Os_sdvig_nagnetatelja_plus.Signaling OR
  protections.Os_sdvig_nagnetatelja_minus.Signaling OR
  protections.Pgaza_na_vyhode_nagnetatelia_GPA_STOP.Signaling OR
  protections.Pgaza_na_vhode_nagnetatelia_GPA_STOP.Signaling OR
  protections.Pgaza_na_vyhode_nagnetatelia.Signaling OR
  protections.dPmaslo_gaz.Signaling OR
  protections.Pmaslo_sm_nizkoe.Signaling OR
  protections.Pmaslo_sm_vysokoe.Signaling OR
  protections.Vibro_skorost_OPED_T1.Signaling OR
  protections.Vibro_skorost_OPED_T2.Signaling OR
  protections.Vibro_skorost_OYP_kolesa_ED_T3.Signaling OR
  protections.Vibro_skorost_OP_kolesa_RH_T4.Signaling OR
  protections.Vibro_skorost_OP_shesterni_RED_T5.Signaling OR
  protections.Vibro_skorost_OP_shesterni_RED_T6.Signaling OR
  protections.dPmaslo_gaz_less100.Signaling OR
  protections.Reg_vozb_off.Signaling OR
  protections.Fail_chastotnii_pusk.Signaling OR
  protections.Off_avar_vikluchatel.Signaling OR
  protections.AOKC_SHKC.Signaling OR
  protections.AO_PRU.Signaling OR
  protections.AO_ot_SHU.Signaling OR
  protections.mvOff.Signaling OR
  protections.Kran1_sdvig.Signaling OR
  protections.Kran2_sdvig.Signaling OR
  protections.Tgaza_na_vyhode_H.Signaling;
END_FUNCTION

FUNCTION nsCepeiUpravlenya : BOOL
  VAR_INPUT
    im : ImConfig;
  END_VAR

  nsCepeiUpravlenya:=
  	im.kran1.So OR im.kran1.Sz OR
  	im.kran2.So OR im.kran2.Sz OR
  	im.kran4.So OR im.kran4.Sz OR
  	im.kran5.So OR im.kran5.Sz OR
  	(*im.kran6.So OR im.kran6.Sz OR*)
  	im.kran3b.So OR im.kran3b.Sz OR
  	im.pns.breakCmdOn OR
  	im.nu1.breakCmdOn OR
  	im.nu2.breakCmdOn OR
  	im.PNS.breakCmdOn OR
            im.v1_Avom.breakCmdOn OR
            im.v2_Avom.breakCmdOn OR
            (*im.Ten.breakCmdOn OR*)
  	im.mv.breakCmdOff;
END_FUNCTION

FUNCTION anyAnalogsPs : BOOL
  VAR_INPUT
    ai : AiConfig;
  END_VAR
  VAR
    statusAi : TYPE_StatusAi;
  END_VAR

  anyAnalogsPs:=
  ai.Toporno_podshipnika_EDT_1.interval= statusAi.HW OR
  ai.Toporno_podshipnika_EDT_1.interval= statusAi.LW OR
  ai.Toy_podshipnika_EDT_2.interval= statusAi.HW OR
  ai.Toy_podshipnika_kol_EDT_3.interval= statusAi.HW OR
  ai.Ty_podshipnika_red_EDT_6.interval= statusAi.HW OR
  ai.Ty_podshipnika_nagnet_EDT_7_1.interval= statusAi.HW OR
  ai.Ty_podshipnika_nagnet_EDT_7_2.interval= statusAi.HW OR
  ai.Toy_podshipnika_svobod_konca_EDT_8_1.interval= statusAi.HW OR
  ai.Toy_podshipnika_svobod_konca_EDT_8_2.interval= statusAi.HW OR
  ai.Tholodnogo_vozduha_ED_kanal_1.interval= statusAi.HW OR
  ai.Tholodnogo_vozduha_ED_kanal_2.interval= statusAi.HW OR
  ai.Tgorjachego_vozduha_ED_kanal_1.interval= statusAi.HW OR
  ai.Tgaza_na_vyhode_H.interval= statusAi.HW OR
  ai.Tmasla_MB.interval= statusAi.LW OR
  ai.Pmasla_posle_GNS.interval= statusAi.LW OR
  ai.Pmasla_posle_NU.interval= statusAi.LW OR
  ai.dPgaza_na_konfuzore.interval= statusAi.HW OR
  ai.Os_sdvig_nagnetatelja_plus.interval= statusAi.HW OR
  ai.Os_sdvig_nagnetatelja_minus.interval= statusAi.HW OR
  ai.dPmaslo_gaz.interval= statusAi.HW OR
  ai.Pgaza_na_vhode_nagnetatelia.interval= statusAi.HW OR
  ai.Pgaza_na_vyhode_nagnetatelia.interval= statusAi.HW OR
  ai.Pimpuls_gaz.interval= statusAi.HW OR
  ai.Pimpuls_gaz.interval= statusAi.LW OR
  ai.Yroven_masla_MB.interval= statusAi.HW OR
  ai.Yroven_masla_MB.interval= statusAi.LW OR
  ai.Tmasla_MB_TEN.interval= statusAi.HW OR
  ai.Tmasla_MB_TEN.interval= statusAi.LW OR
  ai.Vibro_skorost_OYP_kolesa_ED_T3.interval= statusAi.HW OR
  ai.Vibro_skorost_OYP_kolesa_ED_T3.interval= statusAi.LW OR
  ai.Vibro_skorost_OP_kolesa_RH_T4.interval= statusAi.HW OR
  ai.Vibro_skorost_OP_kolesa_RH_T4.interval= statusAi.LW;
END_FUNCTION

FUNCTION analogsNS : BOOL
  VAR_INPUT
    ai : AiConfig;
  END_VAR
  VAR
    statusAi : TYPE_StatusAi;
  END_VAR

  analogsNS:=
    ((ai.Tstali_statora_kanal_1.Interval < statusAi.Normal) AND NOT ai.Tstali_statora_kanal_1.remont)
  OR((ai.Tstali_statora_kanal_2.Interval < statusAi.Normal) AND NOT ai.Tstali_statora_kanal_2.remont)
  OR((ai.Tstali_statora_kanal_3.Interval < statusAi.Normal) AND NOT ai.Tstali_statora_kanal_3.remont)
  OR((ai.Tmedi_statora_kanal_1.Interval < statusAi.Normal) AND NOT ai.Tmedi_statora_kanal_1.remont)
  OR((ai.Tmedi_statora_kanal_2.Interval < statusAi.Normal) AND NOT ai.Tmedi_statora_kanal_2.remont)
  OR((ai.Tmedi_statora_kanal_3.Interval < statusAi.Normal) AND NOT ai.Tmedi_statora_kanal_3.remont)
  OR((ai.Toporno_podshipnika_EDT_1.Interval < statusAi.Normal) AND NOT ai.Toporno_podshipnika_EDT_1.remont)
  OR((ai.Toy_podshipnika_EDT_2.Interval < statusAi.Normal) AND NOT ai.Toy_podshipnika_EDT_2.remont)
  OR((ai.Toy_podshipnika_kol_EDT_3.Interval < statusAi.Normal) AND NOT ai.Toy_podshipnika_kol_EDT_3.remont)
  OR((ai.Toy_podshipnika_kol_EDT_4.Interval < statusAi.Normal) AND NOT ai.Toy_podshipnika_kol_EDT_4.remont)
  OR((ai.Toy_podshipnika_shest_red_EDT_5.Interval < statusAi.Normal) AND NOT ai.Toy_podshipnika_shest_red_EDT_5.remont)
  OR((ai.Ty_podshipnika_red_EDT_6.Interval < statusAi.Normal) AND NOT ai.Ty_podshipnika_red_EDT_6.remont)
  OR((ai.Ty_podshipnika_nagnet_EDT_7_1.Interval < statusAi.Normal) AND NOT ai.Ty_podshipnika_nagnet_EDT_7_1.remont)
  OR((ai.Ty_podshipnika_nagnet_EDT_7_2.Interval < statusAi.Normal) AND NOT ai.Ty_podshipnika_nagnet_EDT_7_2.remont)
  OR((ai.Toy_podshipnika_svobod_konca_EDT_8_1.Interval < statusAi.Normal) AND NOT ai.Toy_podshipnika_svobod_konca_EDT_8_1.remont)
  OR((ai.Toy_podshipnika_svobod_konca_EDT_8_2.Interval < statusAi.Normal) AND NOT ai.Toy_podshipnika_svobod_konca_EDT_8_2.remont)
  OR((ai.Tholodnogo_vozduha_ED_kanal_1.Interval < statusAi.Normal) AND NOT ai.Tholodnogo_vozduha_ED_kanal_1.remont)
  OR((ai.Tholodnogo_vozduha_ED_kanal_2.Interval < statusAi.Normal) AND NOT ai.Tholodnogo_vozduha_ED_kanal_2.remont)
  OR((ai.Tgorjachego_vozduha_ED_kanal_1.Interval < statusAi.Normal) AND NOT ai.Tgorjachego_vozduha_ED_kanal_1.remont)
  OR((ai.Tgorjachego_vozduha_ED_kanal_2.Interval < statusAi.Normal) AND NOT ai.Tgorjachego_vozduha_ED_kanal_2.remont)
  OR((ai.Tnarujnogo_vozduha.Interval < statusAi.Normal) AND NOT ai.Tnarujnogo_vozduha.remont)
  OR((ai.Tgaza_na_vhode_H.Interval < statusAi.Normal) AND NOT ai.Tgaza_na_vhode_H.remont)
  OR((ai.Tgaza_na_vyhode_H.Interval < statusAi.Normal) AND NOT ai.Tgaza_na_vyhode_H.remont)
  OR((ai.Tmasla_posle_AVOM.Interval < statusAi.Normal) AND NOT ai.Tmasla_posle_AVOM.remont)
  OR((ai.Tgorjachego_vozduha_ED_kanal_2.Interval < statusAi.Normal) AND NOT ai.Tgorjachego_vozduha_ED_kanal_2.remont)
  OR((ai.Tmasla_MB.Interval < statusAi.Normal) AND NOT ai.Tmasla_MB.remont)
  OR((ai.dPgaza_na_konfuzore.Interval < statusAi.Normal) AND NOT ai.dPgaza_na_konfuzore.remont)
  OR((ai.Pmaslo_sm_nizkoe.Interval < statusAi.Normal) AND NOT ai.Pmaslo_sm_nizkoe.remont)
  OR((ai.dPgaza_na_maslo_filtre.Interval < statusAi.Normal) AND NOT ai.dPgaza_na_maslo_filtre.remont)
  OR((ai.Pmaslo_sm_vysokoe.Interval < statusAi.Normal) AND NOT ai.Pmaslo_sm_vysokoe.remont)
  OR((ai.Pmasla_posle_GNS.Interval < statusAi.Normal) AND NOT ai.Pmasla_posle_GNS.remont)
  OR((ai.Pmasla_posle_NU.Interval < statusAi.Normal) AND NOT ai.Pmasla_posle_NU.remont)
  OR((ai.Os_sdvig_nagnetatelja_plus.Interval < statusAi.Normal) AND NOT ai.Os_sdvig_nagnetatelja_plus.remont)
  OR((ai.Os_sdvig_nagnetatelja_minus.Interval < statusAi.Normal) AND NOT ai.Os_sdvig_nagnetatelja_minus.remont)
  OR((ai.dPmaslo_gaz.Interval < statusAi.Normal) AND NOT ai.dPmaslo_gaz.remont)
  OR((ai.Pgaza_na_vhode_nagnetatelia.Interval < statusAi.Normal) AND NOT ai.Pgaza_na_vhode_nagnetatelia.remont)
  OR((ai.Pgaza_na_vyhode_nagnetatelia.Interval < statusAi.Normal) AND NOT ai.Pgaza_na_vyhode_nagnetatelia.remont)
  OR((ai.Pimpuls_gaz.Interval < statusAi.Normal) AND NOT ai.Pimpuls_gaz.remont)
  OR((ai.Yroven_masla_MB.Interval < statusAi.Normal) AND NOT ai.Yroven_masla_MB.remont)
  OR((ai.Kontrol_per_220V.Interval < statusAi.Normal) AND NOT ai.Kontrol_per_220V.remont)
  OR((ai.Kontrol_post_220V.Interval < statusAi.Normal) AND NOT ai.Kontrol_post_220V.remont)
  OR((ai.Kontrol_post_220V.Interval < statusAi.Normal) AND NOT ai.Kontrol_post_220V.remont)
  OR((ai.Vibro_skorost_OPED_T1.Interval < statusAi.Normal) AND NOT ai.Vibro_skorost_OPED_T1.remont)
  OR((ai.Vibro_skorost_OYP_kolesa_ED_T3.Interval < statusAi.Normal) AND NOT ai.Vibro_skorost_OYP_kolesa_ED_T3.remont)
  OR((ai.Vibro_skorost_OP_kolesa_RH_T4.Interval < statusAi.Normal) AND NOT ai.Vibro_skorost_OP_kolesa_RH_T4.remont);
END_FUNCTION

FUNCTION_BLOCK ppuAlg
  VAR_IN_OUT
    StrAlg : struct_Alg;
  END_VAR
  VAR
    BMP_Err : struct_PhaseAlgoritm;
    Level_masla_Norm : struct_PhaseAlgoritm;
    T_masla_Norm : struct_PhaseAlgoritm;
    Krans_ready_to_move : struct_PhaseAlgoritm;
  END_VAR
  VAR_IN_OUT
    Krans_Poloj : struct_PhaseAlgoritm;
    Net_AO_KC_SHKS04M : struct_PhaseAlgoritm;
    EGPA_Stop : struct_PhaseAlgoritm;
    Avt_SHU_vkl : struct_PhaseAlgoritm;
    All_IM_Off : struct_PhaseAlgoritm;
    Nalichie220_SHU_Ai : struct_PhaseAlgoritm;
    BP_Norm : struct_PhaseAlgoritm;
    Naprajenie_U_IM : struct_PhaseAlgoritm;
    MV_Poloj_RolledON : struct_PhaseAlgoritm;
    MV_Poloj_RolledOFF : struct_PhaseAlgoritm;
    NOTAnalogNS : struct_PhaseAlgoritm;
    Net_ASPS_Analogs : struct_PhaseAlgoritm;
    Not_AS : struct_PhaseAlgoritm;
    Gotov_Vozb : struct_PhaseAlgoritm;
    Reactornyi_P : struct_PhaseAlgoritm;
    Chastotnyi_P : struct_PhaseAlgoritm;
    dP_kr1 : struct_PhaseAlgoritm;
    Auto_Rej : struct_PhaseAlgoritm;
    CK_IM_Norm : struct_PhaseAlgoritm;
    HAnd_Mode : struct_PhaseAlgoritm;
    Impuls_Gaz : struct_PhaseAlgoritm;
  END_VAR
  VAR
    fb_BMP_Err : fb_ph_CustomPhase;
    fb_Level_masla_Norm : fb_ph_CustomPhase;
    fb_T_masla_Norm : fb_ph_CustomPhase;
    fb_Krans_ready_to_move : fb_ph_CustomPhase;
    fb_Krans_Poloj : fb_ph_CustomPhase;
    fb_Net_AO_KC_SHKS04M : fb_ph_CustomPhase;
    fb_EGPA_Stop : fb_ph_CustomPhase;
    fb_Avt_SHU_vkl : fb_ph_CustomPhase;
    fb_All_IM_Off : fb_ph_CustomPhase;
    fb_Nalichie220_SHU_Ai : fb_ph_CustomPhase;
    fb_BP_Norm : fb_ph_CustomPhase;
    fb_Naprajenie_U_IM : fb_ph_CustomPhase;
    fb_MV_Poloj_RolledON : fb_ph_CustomPhase;
    fb_MV_Poloj_RolledOFF : fb_ph_CustomPhase;
    fb_NOTAnalogNS : fb_ph_CustomPhase;
    fb_Net_ASPS_Analogs : fb_ph_CustomPhase;
    fb_Not_AS : fb_ph_CustomPhase;
    fb_Gotov_Vozb : fb_ph_CustomPhase;
    fb_Reactornyi_P : fb_ph_CustomPhase;
    fb_Chastotnyi_P : fb_ph_CustomPhase;
    fb_dP_kr1 : fb_ph_CustomPhase;
    fb_Auto_Rej : fb_ph_CustomPhase;
    fb_CK_IM_Norm : fb_ph_CustomPhase;
    fb_HAnd_Mode : fb_ph_CustomPhase;
    fb_Impuls_Gaz : fb_ph_CustomPhase;
    _sunpackerCommand : fb_sunpackerCommand;
    modeR_Trig : R_TRIG;
    modeF_Trig : F_TRIG;
    _statusAi : TYPE_StatusAi;
    _Answers : TYPE_Answers;
    _statusDualInput : TYPE_statusDualInput;
    _DualStateImAction : TYPE_DualStateImAction;
    _PhaseAlgoritmAction : TYPE_PhaseAlgoritmAction;
    _basketStats : TYPE_basketStats;
  END_VAR
  VAR_OUTPUT
    puskAllowed : BOOL;
    testAllowed : BOOL;
  END_VAR
  VAR
    ppuDone : BOOL;
    source : BYTE;
    cmd : BYTE;
    lastCmd : BYTE;
    source_for_Status : BYTE;
    cmd_for_Status : BYTE;
    command_error_for_Status : BYTE;
    resetCmdTimer : TON;
    resetCmdTimerPriznak : BOOL;
    onInit : BOOL;
  END_VAR
  VAR_EXTERNAL
    IM : ImConfig;
    ai : AiConfig;
    di : DiConfig;
    algManager : struct_AlgoritmsManager;
    protectManager : struct_ProtectionsManager;
    NotHasRezervNU : BOOL;
    ModeGpa : TYPE_ModeGpa;
    algoritms : AlgoritmsConfig;
  END_VAR

  IF NOT onInit THEN

      fb_BMP_Err(phaseNumber:=0);
      fb_Level_masla_Norm(phaseNumber:=1);
      fb_T_masla_Norm(phaseNumber:=2);
      fb_Krans_ready_to_move(phaseNumber:=5);
      fb_Krans_Poloj(phaseNumber:=6);
      fb_Net_AO_KC_SHKS04M(phaseNumber:=7);
      fb_EGPA_Stop(phaseNumber:=9);
      fb_Avt_SHU_vkl(phaseNumber:=10);
      fb_All_IM_Off(phaseNumber:=11);
      fb_Nalichie220_SHU_Ai(phaseNumber:=12);
      fb_BP_Norm(phaseNumber:=13);
      fb_Naprajenie_U_IM(phaseNumber:=14);
      fb_MV_Poloj_RolledON(phaseNumber:=15);
      fb_MV_Poloj_RolledOFF(phaseNumber:=16);
      fb_NOTAnalogNS(phaseNumber:=17);
      fb_Net_ASPS_Analogs(phaseNumber:=18);
      fb_Not_AS(phaseNumber:=19);
      fb_Gotov_Vozb(phaseNumber:=20);
      fb_Reactornyi_P(phaseNumber:=21);
      fb_Chastotnyi_P(phaseNumber:=22);
      fb_dP_kr1(phaseNumber:=23);
      fb_Auto_Rej(phaseNumber:=24);
      fb_CK_IM_Norm(phaseNumber:=25);
      fb_HAnd_Mode(phaseNumber:=26);
      fb_Impuls_Gaz(phaseNumber:=27);

  onInit:=TRUE;
  END_IF;

  fb_BMP_Err(StrPh:=BMP_Err);
  fb_Level_masla_Norm(StrPh:=Level_masla_Norm);
  fb_T_masla_Norm(StrPh:=T_masla_Norm);
  fb_Krans_ready_to_move(StrPh:=Krans_ready_to_move);
  fb_Krans_Poloj(StrPh:=Krans_Poloj);
  fb_Net_AO_KC_SHKS04M(StrPh:=Net_AO_KC_SHKS04M);
  fb_EGPA_Stop(StrPh:=EGPA_Stop);
  fb_Avt_SHU_vkl(StrPh:=Avt_SHU_vkl);
  fb_All_IM_Off(StrPh:=All_IM_Off);
  fb_Nalichie220_SHU_Ai(StrPh:=Nalichie220_SHU_Ai);
  fb_BP_Norm(StrPh:=BP_Norm);
  fb_Naprajenie_U_IM(StrPh:=Naprajenie_U_IM);
  fb_MV_Poloj_RolledON(StrPh:=MV_Poloj_RolledON);
  fb_MV_Poloj_RolledOFF(StrPh:=MV_Poloj_RolledOFF);
  fb_NOTAnalogNS(StrPh:=NOTAnalogNS);
  fb_Net_ASPS_Analogs(StrPh:=Net_ASPS_Analogs);
  fb_Not_AS(StrPh:=Not_AS);
  fb_Gotov_Vozb(StrPh:=Gotov_Vozb);
  fb_Reactornyi_P(StrPh:=Reactornyi_P);
  fb_Chastotnyi_P(StrPh:=Chastotnyi_P);
  fb_dP_kr1(StrPh:=dP_kr1);
  fb_Auto_Rej(StrPh:=Auto_Rej);
  fb_CK_IM_Norm(StrPh:=CK_IM_Norm);
  fb_HAnd_Mode(StrPh:=HAnd_Mode);
  fb_Impuls_Gaz(StrPh:=Impuls_Gaz);

  IF StrAlg.isRuning THEN

      (*BMP_Err.top:= ((BMPERR_k = 0) OR (kontroller.imit)); надо разобраться кто такой BMPERR_k*)
      (*уровень масла в норме*)
      Level_masla_Norm.top := (ai.Yroven_masla_MB.interval = _statusAi.normal);

      (*температура масла в норме*)
      T_masla_Norm.top:= (ai.Tmasla_MB.interval = _statusAi.normal);

      (*kраны готовы к управлению*)
      Krans_ready_to_move.top:= NOT (IM.Kran1.So OR IM.Kran1.Sz OR IM.Kran2.So OR IM.Kran2.Sz OR IM.Kran3.So OR
                                     IM.Kran3.Sz OR IM.Kran3b.So OR IM.Kran3b.Sz OR IM.Kran4.So OR IM.Kran4.Sz OR
  			     IM.Kran5.So OR IM.Kran5.Sz OR IM.Kran6.So OR IM.Kran6.Sz);

      (*положение кранов верное*)
      Krans_Poloj.top:= (Im.Kran1.onStatus=_statusDualInput.STATUS_OFF) AND
  		  (Im.Kran2.onStatus=_statusDualInput.STATUS_OFF) AND
  		  (Im.Kran3.onStatus=_statusDualInput.STATUS_OFF) AND
  		  (Im.Kran3b.onStatus=_statusDualInput.STATUS_ON) AND
  		  (Im.Kran4.onStatus=_statusDualInput.STATUS_OFF) AND
  		  (Im.Kran5.onStatus=_statusDualInput.STATUS_ON) AND
                        (Im.Kran6.onStatus=_statusDualInput.STATUS_ON);
      (*Нет АО от ШКС
      Net_AO_KC_SHKS04M.top:= haveAlarms(); кто такой haveAlarms*)
